LIN {X 0,Y 502.812,Z 410.918,A -85,B 0,C 180,E1 -5734.96,E2 -5734.96} C_VEL
LIN {X 0,Y 504.611,Z 420.54,A -85,B 0,C 180,E1 -5736.546,E2 -5736.546} C_VEL
LIN {X 0,Y 504.361,Z 436.32,A -85,B 0,C 180,E1 -5739.005,E2 -5739.005} C_VEL
LIN {X 0,Y 503.884,Z 455.526,A -85,B 0,C 180,E1 -5741.972,E2 -5741.972} C_VEL
LIN {X 0,Y 503.523,Z 470.549,A -85,B 0,C 180,E1 -5744.274,E2 -5744.274} C_VEL
LIN {X 0,Y 505.329,Z 482.17,A -85,B 0,C 180,E1 -5744.511,E2 -5744.511} C_VEL
LIN {X 0,Y 504.68,Z 580.109,A -85,B 0,C 180,E1 -5745.998,E2 -5745.998} C_VEL
LIN {X 0,Y 504.442,Z 593.546,A -85,B 0,C 180,E1 -5746.376,E2 -5746.376} C_VEL
LIN {X 0,Y 504.146,Z 606.339,A -85,B 0,C 180,E1 -5746.907,E2 -5746.907} C_VEL
LIN {X 0,Y 503.865,Z 618.187,A -85,B 0,C 180,E1 -5747.573,E2 -5747.573} C_VEL
LIN {X 0,Y 503.569,Z 628.743,A -85,B 0,C 180,E1 -5748.324,E2 -5748.324} C_VEL
LIN {X 0,Y 503.221,Z 639.022,A -85,B 0,C 180,E1 -5749.234,E2 -5749.234} C_VEL
LIN {X 0,Y 502.902,Z 649.127,A -85,B 0,C 180,E1 -5750.346,E2 -5750.346} C_VEL
LIN {X 0,Y 502.609,Z 657.945,A -85,B 0,C 180,E1 -5751.557,E2 -5751.557} C_VEL
LIN {X 0,Y 502.408,Z 665.014,A -85,B 0,C 180,E1 -5752.767,E2 -5752.767} C_VEL
LIN {X 0,Y 502.316,Z 670.67,A -85,B 0,C 180,E1 -5753.977,E2 -5753.977} C_VEL
LIN {X 0,Y 502.118,Z 675.083,A -85,B 0,C 180,E1 -5755.183,E2 -5755.183} C_VEL
LIN {X 0,Y 502.218,Z 677.414,A -85,B 0,C 180,E1 -5755.988,E2 -5755.988} C_VEL
LIN {X 0,Y 502.124,Z 679.291,A -85,B 0,C 180,E1 -5756.791,E2 -5756.791} C_VEL
LIN {X 0,Y 502.121,Z 680.748,A -85,B 0,C 180,E1 -5757.593,E2 -5757.593} C_VEL
LIN {X 0,Y 502.036,Z 681.79,A -85,B 0,C 180,E1 -5758.396,E2 -5758.396} C_VEL
LIN {X 0,Y 501.98,Z 682.648,A -85,B 0,C 180,E1 -5760,E2 -5760} C_VEL
LIN {X 0,Y 501.99,Z 682.478,A -85,B 0,C 180,E1 -5760.802,E2 -5760.802} C_VEL
LIN {X 0,Y 502.037,Z 681.897,A -85,B 0,C 180,E1 -5761.604,E2 -5761.604} C_VEL
LIN {X 0,Y 502.121,Z 680.912,A -85,B 0,C 180,E1 -5762.407,E2 -5762.407} C_VEL
LIN {X 0,Y 502.125,Z 679.521,A -85,B 0,C 180,E1 -5763.209,E2 -5763.209} C_VEL
LIN {X 0,Y 502.188,Z 676.607,A -85,B 0,C 180,E1 -5764.414,E2 -5764.414} C_VEL
LIN {X 0,Y 502.289,Z 672.64,A -85,B 0,C 180,E1 -5765.621,E2 -5765.621} C_VEL
LIN {X 0,Y 502.369,Z 666.641,A -85,B 0,C 180,E1 -5767.011,E2 -5767.011} C_VEL
LIN {X 0,Y 502.552,Z 659.852,A -85,B 0,C 180,E1 -5768.241,E2 -5768.241} C_VEL
LIN {X 0,Y 502.792,Z 651.442,A -85,B 0,C 180,E1 -5769.453,E2 -5769.453} C_VEL
LIN {X 0,Y 503.042,Z 642.838,A -85,B 0,C 180,E1 -5770.464,E2 -5770.464} C_VEL
LIN {X 0,Y 503.426,Z 632.166,A -85,B 0,C 180,E1 -5771.475,E2 -5771.475} C_VEL
LIN {X 0,Y 503.752,Z 621.087,A -85,B 0,C 180,E1 -5772.316,E2 -5772.316} C_VEL
LIN {X 0,Y 504.055,Z 609.692,A -85,B 0,C 180,E1 -5772.993,E2 -5772.993} C_VEL
LIN {X 0,Y 504.289,Z 597.377,A -85,B 0,C 180,E1 -5773.551,E2 -5773.551} C_VEL
LIN {X 0,Y 504.521,Z 584.764,A -85,B 0,C 180,E1 -5773.955,E2 -5773.955} C_VEL
LIN {X 0,Y 504.744,Z 570.118,A -85,B 0,C 180,E1 -5774.232,E2 -5774.232} C_VEL
LIN {X 0,Y 505.211,Z 480.854,A -85,B 0,C 180,E1 -5775.591,E2 -5775.591} C_VEL
LIN {X 0,Y 503.576,Z 470.754,A -85,B 0,C 180,E1 -5775.817,E2 -5775.817} C_VEL
LIN {X 0,Y 503.993,Z 450.167,A -85,B 0,C 180,E1 -5778.918,E2 -5778.918} C_VEL
LIN {X 0,Y 504.321,Z 430.326,A -85,B 0,C 180,E1 -5781.887,E2 -5781.887} C_VEL
LIN {X 0,Y 504.447,Z 419.832,A -85,B 0,C 180,E1 -5783.429,E2 -5783.429} C_VEL
LIN {X 0,Y 502.802,Z 410.856,A -85,B 0,C 180,E1 -5784.848,E2 -5784.848} C_VEL
LIN {X 0,Y 502.779,Z 410.86,A -85,B 0,C 180,E1 -5787.47,E2 -5787.47} C_VEL
LIN {X 0,Y 502.805,Z 410.855,A -85,B 0,C 180,E1 -5790.212,E2 -5790.212} C_VEL
LIN {X 0,Y 502.834,Z 410.851,A -85,B 0,C 180,E1 -5793.031,E2 -5793.031} C_VEL
LIN {X 0,Y 502.77,Z 410.856,A -85,B 0,C 180,E1 -5795.952,E2 -5795.952} C_VEL
LIN {X 0,Y 502.803,Z 410.855,A -85,B 0,C 180,E1 -5798.976,E2 -5798.976} C_VEL
LIN {X 0,Y 502.798,Z 410.852,A -85,B 0,C 180,E1 -5802.139,E2 -5802.139} C_VEL
LIN {X 0,Y 502.804,Z 410.854,A -85,B 0,C 180,E1 -5805.468,E2 -5805.468} C_VEL
LIN {X 0,Y 502.822,Z 410.853,A -85,B 0,C 180,E1 -5808.934,E2 -5808.934} C_VEL
LIN {X 0,Y 502.793,Z 410.852,A -85,B 0,C 180,E1 -5812.046,E2 -5812.046} C_VEL
LIN {X 0,Y 502.8,Z 410.854,A -85,B 0,C 180,E1 -5815.034,E2 -5815.034} C_VEL
LIN {X 0,Y 502.785,Z 410.855,A -85,B 0,C 180,E1 -5817.915,E2 -5817.915} C_VEL
LIN {X 0,Y 502.806,Z 410.856,A -85,B 0,C 180,E1 -5820.711,E2 -5820.711} C_VEL
LIN {X 0,Y 502.835,Z 411.023,A -85,B 0,C 180,E1 -5822.336,E2 -5822.336} C_VEL
LIN {X 0,Y 505.373,Z 423.463,A -85,B 0,C 180,E1 -5824.241,E2 -5824.241} C_VEL
LIN {X 0,Y 504.875,Z 441.29,A -85,B 0,C 180,E1 -5826.743,E2 -5826.743} C_VEL
LIN {X 0,Y 504.364,Z 458.409,A -85,B 0,C 180,E1 -5829.112,E2 -5829.112} C_VEL
LIN {X 0,Y 503.788,Z 480.465,A -85,B 0,C 180,E1 -5832.127,E2 -5832.127} C_VEL
LIN {X 0,Y 503.365,Z 495.682,A -85,B 0,C 180,E1 -5834.186,E2 -5834.186} C_VEL
LIN {X 0,Y 505.216,Z 510.923,A -85,B 0,C 180,E1 -5834.498,E2 -5834.498} C_VEL
LIN {X 0,Y 504.735,Z 596.683,A -85,B 0,C 180,E1 -5835.768,E2 -5835.768} C_VEL
LIN {X 0,Y 504.502,Z 611.005,A -85,B 0,C 180,E1 -5836.044,E2 -5836.044} C_VEL
LIN {X 0,Y 504.216,Z 624.892,A -85,B 0,C 180,E1 -5836.499,E2 -5836.499} C_VEL
LIN {X 0,Y 503.892,Z 635.855,A -85,B 0,C 180,E1 -5837.003,E2 -5837.003} C_VEL
LIN {X 0,Y 503.617,Z 646.876,A -85,B 0,C 180,E1 -5837.649,E2 -5837.649} C_VEL
LIN {X 0,Y 503.303,Z 657.249,A -85,B 0,C 180,E1 -5838.42,E2 -5838.42} C_VEL
LIN {X 0,Y 502.974,Z 667.319,A -85,B 0,C 180,E1 -5839.331,E2 -5839.331} C_VEL
LIN {X 0,Y 502.708,Z 676.4,A -85,B 0,C 180,E1 -5840.342,E2 -5840.342} C_VEL
LIN {X 0,Y 502.53,Z 683.874,A -85,B 0,C 180,E1 -5841.353,E2 -5841.353} C_VEL
LIN {X 0,Y 502.351,Z 691.292,A -85,B 0,C 180,E1 -5842.564,E2 -5842.564} C_VEL
LIN {X 0,Y 502.235,Z 696.303,A -85,B 0,C 180,E1 -5843.572,E2 -5843.572} C_VEL
LIN {X 0,Y 502.184,Z 701.137,A -85,B 0,C 180,E1 -5844.781,E2 -5844.781} C_VEL
LIN {X 0,Y 502.231,Z 704.816,A -85,B 0,C 180,E1 -5845.988,E2 -5845.988} C_VEL
LIN {X 0,Y 502.206,Z 706.732,A -85,B 0,C 180,E1 -5846.791,E2 -5846.791} C_VEL
LIN {X 0,Y 502.124,Z 708.179,A -85,B 0,C 180,E1 -5847.593,E2 -5847.593} C_VEL
LIN {X 0,Y 502.041,Z 709.755,A -85,B 0,C 180,E1 -5849.198,E2 -5849.198} C_VEL
LIN {X 0,Y 502.04,Z 709.991,A -85,B 0,C 180,E1 -5850,E2 -5850} C_VEL
LIN {X 0,Y 502.041,Z 709.76,A -85,B 0,C 180,E1 -5850.802,E2 -5850.802} C_VEL
LIN {X 0,Y 502.065,Z 709.113,A -85,B 0,C 180,E1 -5851.604,E2 -5851.604} C_VEL
LIN {X 0,Y 502.206,Z 706.61,A -85,B 0,C 180,E1 -5853.209,E2 -5853.209} C_VEL
LIN {X 0,Y 502.202,Z 703.539,A -85,B 0,C 180,E1 -5854.414,E2 -5854.414} C_VEL
LIN {X 0,Y 502.272,Z 699.389,A -85,B 0,C 180,E1 -5855.621,E2 -5855.621} C_VEL
LIN {X 0,Y 502.316,Z 694.249,A -85,B 0,C 180,E1 -5856.79,E2 -5856.79} C_VEL
LIN {X 0,Y 502.403,Z 688.572,A -85,B 0,C 180,E1 -5857.839,E2 -5857.839} C_VEL
LIN {X 0,Y 502.585,Z 682.001,A -85,B 0,C 180,E1 -5858.848,E2 -5858.848} C_VEL
LIN {X 0,Y 502.79,Z 674.116,A -85,B 0,C 180,E1 -5859.859,E2 -5859.859} C_VEL
LIN {X 0,Y 503.073,Z 664.588,A -85,B 0,C 180,E1 -5860.871,E2 -5860.871} C_VEL
LIN {X 0,Y 503.361,Z 655.159,A -85,B 0,C 180,E1 -5861.68,E2 -5861.68} C_VEL
LIN {X 0,Y 503.524,Z 645.309,A -85,B 0,C 180,E1 -5862.381,E2 -5862.381} C_VEL
LIN {X 0,Y 503.86,Z 633.683,A -85,B 0,C 180,E1 -5863.049,E2 -5863.049} C_VEL
LIN {X 0,Y 504.154,Z 622.054,A -85,B 0,C 180,E1 -5863.555,E2 -5863.555} C_VEL
LIN {X 0,Y 504.488,Z 608.94,A -85,B 0,C 180,E1 -5863.956,E2 -5863.956} C_VEL
LIN {X 0,Y 504.652,Z 593.561,A -85,B 0,C 180,E1 -5864.234,E2 -5864.234} C_VEL
LIN {X 0,Y 505.203,Z 510.39,A -85,B 0,C 180,E1 -5865.485,E2 -5865.485} C_VEL
LIN {X 0,Y 503.281,Z 493.921,A -85,B 0,C 180,E1 -5865.828,E2 -5865.828} C_VEL
LIN {X 0,Y 503.793,Z 470.715,A -85,B 0,C 180,E1 -5868.926,E2 -5868.926} C_VEL
LIN {X 0,Y 504.326,Z 447.248,A -85,B 0,C 180,E1 -5872.102,E2 -5872.102} C_VEL
LIN {X 0,Y 504.989,Z 424.658,A -85,B 0,C 180,E1 -5875.228,E2 -5875.228} C_VEL
LIN {X 0,Y 504.522,Z 419.183,A -85,B 0,C 180,E1 -5876.027,E2 -5876.027} C_VEL
LIN {X 0,Y 502.809,Z 410.856,A -85,B 0,C 180,E1 -5877.311,E2 -5877.311} C_VEL
LIN {X 0,Y 502.805,Z 410.856,A -85,B 0,C 180,E1 -5880.212,E2 -5880.212} C_VEL
LIN {X 0,Y 502.834,Z 410.851,A -85,B 0,C 180,E1 -5883.031,E2 -5883.031} C_VEL
LIN {X 0,Y 502.769,Z 410.858,A -85,B 0,C 180,E1 -5885.952,E2 -5885.952} C_VEL
LIN {X 0,Y 502.803,Z 410.854,A -85,B 0,C 180,E1 -5888.976,E2 -5888.976} C_VEL
LIN {X 0,Y 502.805,Z 410.85,A -85,B 0,C 180,E1 -5892.199,E2 -5892.199} C_VEL
LIN {X 0,Y 502.804,Z 410.856,A -85,B 0,C 180,E1 -5895.468,E2 -5895.468} C_VEL
LIN {X 0,Y 502.822,Z 410.853,A -85,B 0,C 180,E1 -5898.934,E2 -5898.934} C_VEL
LIN {X 0,Y 502.796,Z 410.851,A -85,B 0,C 180,E1 -5902.046,E2 -5902.046} C_VEL
LIN {X 0,Y 502.803,Z 410.857,A -85,B 0,C 180,E1 -5905.034,E2 -5905.034} C_VEL
LIN {X 0,Y 502.786,Z 410.853,A -85,B 0,C 180,E1 -5907.915,E2 -5907.915} C_VEL
LIN {X 0,Y 502.825,Z 410.854,A -85,B 0,C 180,E1 -5910.712,E2 -5910.712} C_VEL
LIN {X 0,Y 502.866,Z 410.845,A -85,B 0,C 180,E1 -5913.439,E2 -5913.439} C_VEL
LIN {X 0,Y 502.779,Z 410.858,A -85,B 0,C 180,E1 -5916.086,E2 -5916.086} C_VEL
LIN {X 0,Y 502.786,Z 410.86,A -85,B 0,C 180,E1 -5918.689,E2 -5918.689} C_VEL
LIN {X 0,Y 502.825,Z 410.851,A -85,B 0,C 180,E1 -5921.248,E2 -5921.248} C_VEL
LIN {X 0,Y 502.835,Z 410.853,A -85,B 0,C 180,E1 -5924.345,E2 -5924.345} C_VEL
LIN {X 0,Y 505.443,Z 418.562,A -85,B 0,C 180,E1 -5924.56,E2 -5924.56} C_VEL
LIN {X 0,Y 504.73,Z 513.794,A -85,B 0,C 180,E1 -5926.051,E2 -5926.051} C_VEL
LIN {X 0,Y 504.537,Z 527.27,A -85,B 0,C 180,E1 -5926.43,E2 -5926.43} C_VEL
LIN {X 0,Y 504.305,Z 539.968,A -85,B 0,C 180,E1 -5926.962,E2 -5926.962} C_VEL
LIN {X 0,Y 504.046,Z 551.757,A -85,B 0,C 180,E1 -5927.631,E2 -5927.631} C_VEL
LIN {X 0,Y 503.743,Z 562.812,A -85,B 0,C 180,E1 -5928.431,E2 -5928.431} C_VEL
LIN {X 0,Y 503.456,Z 572.863,A -85,B 0,C 180,E1 -5929.341,E2 -5929.341} C_VEL
LIN {X 0,Y 503.173,Z 581.893,A -85,B 0,C 180,E1 -5930.351,E2 -5930.351} C_VEL
LIN {X 0,Y 502.846,Z 590.669,A -85,B 0,C 180,E1 -5931.561,E2 -5931.561} C_VEL
LIN {X 0,Y 502.642,Z 597.668,A -85,B 0,C 180,E1 -5932.771,E2 -5932.771} C_VEL
LIN {X 0,Y 502.535,Z 603.214,A -85,B 0,C 180,E1 -5933.979,E2 -5933.979} C_VEL
LIN {X 0,Y 502.328,Z 607.57,A -85,B 0,C 180,E1 -5935.185,E2 -5935.185} C_VEL
LIN {X 0,Y 502.363,Z 609.847,A -85,B 0,C 180,E1 -5935.989,E2 -5935.989} C_VEL
LIN {X 0,Y 502.26,Z 611.712,A -85,B 0,C 180,E1 -5936.791,E2 -5936.791} C_VEL
LIN {X 0,Y 502.166,Z 613.13,A -85,B 0,C 180,E1 -5937.594,E2 -5937.594} C_VEL
LIN {X 0,Y 502.085,Z 614.717,A -85,B 0,C 180,E1 -5939.198,E2 -5939.198} C_VEL
LIN {X 0,Y 502.079,Z 614.934,A -85,B 0,C 180,E1 -5940,E2 -5940} C_VEL
LIN {X 0,Y 502.082,Z 614.729,A -85,B 0,C 180,E1 -5940.802,E2 -5940.802} C_VEL
LIN {X 0,Y 502.152,Z 613.119,A -85,B 0,C 180,E1 -5942.406,E2 -5942.406} C_VEL
LIN {X 0,Y 502.256,Z 611.723,A -85,B 0,C 180,E1 -5943.209,E2 -5943.209} C_VEL
LIN {X 0,Y 502.359,Z 608.801,A -85,B 0,C 180,E1 -5944.413,E2 -5944.413} C_VEL
LIN {X 0,Y 502.343,Z 604.86,A -85,B 0,C 180,E1 -5945.62,E2 -5945.62} C_VEL
LIN {X 0,Y 502.52,Z 598.883,A -85,B 0,C 180,E1 -5947.004,E2 -5947.004} C_VEL
LIN {X 0,Y 502.77,Z 592.082,A -85,B 0,C 180,E1 -5948.238,E2 -5948.238} C_VEL
LIN {X 0,Y 502.992,Z 583.786,A -85,B 0,C 180,E1 -5949.449,E2 -5949.449} C_VEL
LIN {X 0,Y 503.332,Z 575.218,A -85,B 0,C 180,E1 -5950.458,E2 -5950.458} C_VEL
LIN {X 0,Y 503.631,Z 564.636,A -85,B 0,C 180,E1 -5951.47,E2 -5951.47} C_VEL
LIN {X 0,Y 503.938,Z 555.004,A -85,B 0,C 180,E1 -5952.216,E2 -5952.216} C_VEL
LIN {X 0,Y 504.182,Z 544.302,A -85,B 0,C 180,E1 -5952.887,E2 -5952.887} C_VEL
LIN {X 0,Y 504.424,Z 532.882,A -85,B 0,C 180,E1 -5953.445,E2 -5953.445} C_VEL
LIN {X 0,Y 504.654,Z 519.828,A -85,B 0,C 180,E1 -5953.9,E2 -5953.9} C_VEL
LIN {X 0,Y 504.785,Z 507.422,A -85,B 0,C 180,E1 -5954.179,E2 -5954.179} C_VEL
LIN {X 0,Y 505.314,Z 418.371,A -85,B 0,C 180,E1 -5955.527,E2 -5955.527} C_VEL
LIN {X 0,Y 502.826,Z 410.854,A -85,B 0,C 180,E1 -5955.73,E2 -5955.73} C_VEL
LIN {X 0,Y 502.814,Z 410.852,A -85,B 0,C 180,E1 -5958.752,E2 -5958.752} C_VEL
LIN {X 0,Y 502.784,Z 410.861,A -85,B 0,C 180,E1 -5961.311,E2 -5961.311} C_VEL
LIN {X 0,Y 502.772,Z 410.854,A -85,B 0,C 180,E1 -5963.915,E2 -5963.915} C_VEL
LIN {X 0,Y 502.839,Z 410.845,A -85,B 0,C 180,E1 -5966.568,E2 -5966.568} C_VEL
LIN {X 0,Y 502.825,Z 410.855,A -85,B 0,C 180,E1 -5969.288,E2 -5969.288} C_VEL
LIN {X 0,Y 502.786,Z 410.848,A -85,B 0,C 180,E1 -5972.085,E2 -5972.085} C_VEL
LIN {X 0,Y 502.802,Z 410.849,A -85,B 0,C 180,E1 -5974.966,E2 -5974.966} C_VEL
LIN {X 0,Y 502.796,Z 410.851,A -85,B 0,C 180,E1 -5977.954,E2 -5977.954} C_VEL
LIN {X 0,Y 502.823,Z 410.85,A -85,B 0,C 180,E1 -5981.066,E2 -5981.066} C_VEL
LIN {X 0,Y 502.767,Z 410.856,A -85,B 0,C 180,E1 -5983.56,E2 -5983.56} C_VEL
LIN {X 0,Y 502.089,Z 410.943,A -85,B 0,C 180,E1 -5984.229,E2 -5984.229} C_VEL
LIN {X 0,Y 499.217,Z 411.293,A -85,B 0,C 180,E1 -5985.314,E2 -5985.314} C_VEL
LIN {X 0,Y 496.809,Z 411.592,A -85,B 0,C 180,E1 -5986.189,E2 -5986.189} C_VEL
LIN {X 0,Y 495.798,Z 411.727,A -85,B 0,C 180,E1 -5986.865,E2 -5986.865} C_VEL
LIN {X 0,Y 495.728,Z 411.735,A -85,B 0,C 180,E1 -5987.094,E2 -5987.094} C_VEL
LIN {X 0,Y 495.761,Z 411.724,A -85,B 0,C 180,E1 -5989.953,E2 -5989.953} C_VEL
LIN {X 0,Y 495.721,Z 411.738,A -85,B 0,C 180,E1 -5992.555,E2 -5992.555} C_VEL
LIN {X 0,Y 495.78,Z 411.725,A -85,B 0,C 180,E1 -5995.457,E2 -5995.457} C_VEL
LIN {X 0,Y 495.757,Z 411.734,A -85,B 0,C 180,E1 -5998.364,E2 -5998.364} C_VEL
LIN {X 0,Y 495.74,Z 411.734,A -85,B 0,C 180,E1 -6001.518,E2 -6001.518} C_VEL
LIN {X 0,Y 495.756,Z 411.755,A -85,B 0,C 180,E1 -6004.775,E2 -6004.775} C_VEL
LIN {X 0,Y 497.706,Z 422.006,A -85,B 0,C 180,E1 -6006.49,E2 -6006.49} C_VEL
LIN {X 0,Y 497.308,Z 438.63,A -85,B 0,C 180,E1 -6009.143,E2 -6009.143} C_VEL
LIN {X 0,Y 496.828,Z 455.991,A -85,B 0,C 180,E1 -6011.868,E2 -6011.868} C_VEL
LIN {X 0,Y 496.586,Z 470.293,A -85,B 0,C 180,E1 -6014.017,E2 -6014.017} C_VEL
LIN {X 0,Y 498.587,Z 482.825,A -85,B 0,C 180,E1 -6014.271,E2 -6014.271} C_VEL
LIN {X 0,Y 497.993,Z 578.618,A -85,B 0,C 180,E1 -6015.675,E2 -6015.675} C_VEL
LIN {X 0,Y 497.758,Z 592.263,A -85,B 0,C 180,E1 -6016.034,E2 -6016.034} C_VEL
LIN {X 0,Y 497.478,Z 604.399,A -85,B 0,C 180,E1 -6016.52,E2 -6016.52} C_VEL
LIN {X 0,Y 497.123,Z 617.014,A -85,B 0,C 180,E1 -6017.208,E2 -6017.208} C_VEL
LIN {X 0,Y 496.84,Z 627.65,A -85,B 0,C 180,E1 -6017.957,E2 -6017.957} C_VEL
LIN {X 0,Y 496.385,Z 638.11,A -85,B 0,C 180,E1 -6018.877,E2 -6018.877} C_VEL
LIN {X 0,Y 495.982,Z 648.406,A -85,B 0,C 180,E1 -6020.004,E2 -6020.004} C_VEL
LIN {X 0,Y 495.678,Z 657.346,A -85,B 0,C 180,E1 -6021.233,E2 -6021.233} C_VEL
LIN {X 0,Y 495.404,Z 664.523,A -85,B 0,C 180,E1 -6022.46,E2 -6022.46} C_VEL
LIN {X 0,Y 495.253,Z 669.395,A -85,B 0,C 180,E1 -6023.481,E2 -6023.481} C_VEL
LIN {X 0,Y 495.128,Z 674.109,A -85,B 0,C 180,E1 -6024.706,E2 -6024.706} C_VEL
LIN {X 0,Y 495.148,Z 677.717,A -85,B 0,C 180,E1 -6025.93,E2 -6025.93} C_VEL
LIN {X 0,Y 495.05,Z 679.577,A -85,B 0,C 180,E1 -6026.745,E2 -6026.745} C_VEL
LIN {X 0,Y 495.025,Z 681.001,A -85,B 0,C 180,E1 -6027.559,E2 -6027.559} C_VEL
LIN {X 0,Y 494.911,Z 682.615,A -85,B 0,C 180,E1 -6029.186,E2 -6029.186} C_VEL
LIN {X 0,Y 494.898,Z 682.853,A -85,B 0,C 180,E1 -6030,E2 -6030} C_VEL
LIN {X 0,Y 494.911,Z 682.667,A -85,B 0,C 180,E1 -6030.814,E2 -6030.814} C_VEL
LIN {X 0,Y 495.025,Z 681.121,A -85,B 0,C 180,E1 -6032.441,E2 -6032.441} C_VEL
LIN {X 0,Y 495.051,Z 679.763,A -85,B 0,C 180,E1 -6033.255,E2 -6033.255} C_VEL
LIN {X 0,Y 495.102,Z 676.905,A -85,B 0,C 180,E1 -6034.478,E2 -6034.478} C_VEL
LIN {X 0,Y 495.234,Z 673.02,A -85,B 0,C 180,E1 -6035.701,E2 -6035.701} C_VEL
LIN {X 0,Y 495.308,Z 667.992,A -85,B 0,C 180,E1 -6036.927,E2 -6036.927} C_VEL
LIN {X 0,Y 495.52,Z 661.646,A -85,B 0,C 180,E1 -6038.154,E2 -6038.154} C_VEL
LIN {X 0,Y 495.766,Z 653.766,A -85,B 0,C 180,E1 -6039.383,E2 -6039.383} C_VEL
LIN {X 0,Y 496.058,Z 645.718,A -85,B 0,C 180,E1 -6040.407,E2 -6040.407} C_VEL
LIN {X 0,Y 496.495,Z 635.844,A -85,B 0,C 180,E1 -6041.43,E2 -6041.43} C_VEL
LIN {X 0,Y 496.888,Z 624.635,A -85,B 0,C 180,E1 -6042.362,E2 -6042.362} C_VEL
LIN {X 0,Y 497.232,Z 613.919,A -85,B 0,C 180,E1 -6043.07,E2 -6043.07} C_VEL
LIN {X 0,Y 497.547,Z 601.827,A -85,B 0,C 180,E1 -6043.686,E2 -6043.686} C_VEL
LIN {X 0,Y 497.877,Z 588.519,A -85,B 0,C 180,E1 -6044.171,E2 -6044.171} C_VEL
LIN {X 0,Y 498.052,Z 576.639,A -85,B 0,C 180,E1 -6044.453,E2 -6044.453} C_VEL
LIN {X 0,Y 498.539,Z 482.079,A -85,B 0,C 180,E1 -6045.832,E2 -6045.832} C_VEL
LIN {X 0,Y 496.57,Z 470.209,A -85,B 0,C 180,E1 -6046.082,E2 -6046.082} C_VEL
LIN {X 0,Y 496.967,Z 451.125,A -85,B 0,C 180,E1 -6048.981,E2 -6048.981} C_VEL
LIN {X 0,Y 497.506,Z 432.156,A -85,B 0,C 180,E1 -6051.984,E2 -6051.984} C_VEL
LIN {X 0,Y 497.746,Z 422.712,A -85,B 0,C 180,E1 -6053.486,E2 -6053.486} C_VEL
LIN {X 0,Y 495.74,Z 411.737,A -85,B 0,C 180,E1 -6055.338,E2 -6055.338} C_VEL
LIN {X 0,Y 495.74,Z 411.732,A -85,B 0,C 180,E1 -6058.482,E2 -6058.482} C_VEL
LIN {X 0,Y 495.757,Z 411.736,A -85,B 0,C 180,E1 -6061.636,E2 -6061.636} C_VEL
LIN {X 0,Y 495.78,Z 411.727,A -85,B 0,C 180,E1 -6064.543,E2 -6064.543} C_VEL
LIN {X 0,Y 495.724,Z 411.737,A -85,B 0,C 180,E1 -6067.562,E2 -6067.562} C_VEL
LIN {X 0,Y 495.769,Z 411.726,A -85,B 0,C 180,E1 -6070.7,E2 -6070.7} C_VEL
LIN {X 0,Y 495.737,Z 411.728,A -85,B 0,C 180,E1 -6074.001,E2 -6074.001} C_VEL
LIN {X 0,Y 495.73,Z 411.734,A -85,B 0,C 180,E1 -6077.117,E2 -6077.117} C_VEL
LIN {X 0,Y 495.762,Z 411.727,A -85,B 0,C 180,E1 -6079.953,E2 -6079.953} C_VEL
LIN {X 0,Y 495.722,Z 411.736,A -85,B 0,C 180,E1 -6082.554,E2 -6082.554} C_VEL
LIN {X 0,Y 495.78,Z 411.724,A -85,B 0,C 180,E1 -6085.457,E2 -6085.457} C_VEL
LIN {X 0,Y 495.757,Z 411.734,A -85,B 0,C 180,E1 -6088.364,E2 -6088.364} C_VEL
LIN {X 0,Y 495.74,Z 411.731,A -85,B 0,C 180,E1 -6091.518,E2 -6091.518} C_VEL
LIN {X 0,Y 495.778,Z 411.816,A -85,B 0,C 180,E1 -6094.776,E2 -6094.776} C_VEL
LIN {X 0,Y 497.561,Z 420.974,A -85,B 0,C 180,E1 -6096.306,E2 -6096.306} C_VEL
LIN {X 0,Y 497.665,Z 427.684,A -85,B 0,C 180,E1 -6097.367,E2 -6097.367} C_VEL
LIN {X 0,Y 497.204,Z 444.245,A -85,B 0,C 180,E1 -6099.954,E2 -6099.954} C_VEL
LIN {X 0,Y 496.748,Z 461.979,A -85,B 0,C 180,E1 -6102.716,E2 -6102.716} C_VEL
LIN {X 0,Y 496.599,Z 470.761,A -85,B 0,C 180,E1 -6104.053,E2 -6104.053} C_VEL
LIN {X 0,Y 498.5,Z 482.776,A -85,B 0,C 180,E1 -6104.306,E2 -6104.306} C_VEL
LIN {X 0,Y 497.776,Z 580.486,A -85,B 0,C 180,E1 -6105.826,E2 -6105.826} C_VEL
LIN {X 0,Y 497.494,Z 593.83,A -85,B 0,C 180,E1 -6106.208,E2 -6106.208} C_VEL
LIN {X 0,Y 497.222,Z 606.079,A -85,B 0,C 180,E1 -6106.721,E2 -6106.721} C_VEL
LIN {X 0,Y 496.876,Z 618.283,A -85,B 0,C 180,E1 -6107.413,E2 -6107.413} C_VEL
LIN {X 0,Y 496.556,Z 629.927,A -85,B 0,C 180,E1 -6108.261,E2 -6108.261} C_VEL
LIN {X 0,Y 496.142,Z 640.999,A -85,B 0,C 180,E1 -6109.285,E2 -6109.285} C_VEL
LIN {X 0,Y 495.799,Z 650.77,A -85,B 0,C 180,E1 -6110.412,E2 -6110.412} C_VEL
LIN {X 0,Y 495.537,Z 659.295,A -85,B 0,C 180,E1 -6111.641,E2 -6111.641} C_VEL
LIN {X 0,Y 495.326,Z 666.262,A -85,B 0,C 180,E1 -6112.889,E2 -6112.889} C_VEL
LIN {X 0,Y 495.229,Z 672.379,A -85,B 0,C 180,E1 -6114.299,E2 -6114.299} C_VEL
LIN {X 0,Y 495.087,Z 676.45,A -85,B 0,C 180,E1 -6115.522,E2 -6115.522} C_VEL
LIN {X 0,Y 495.05,Z 679.461,A -85,B 0,C 180,E1 -6116.745,E2 -6116.745} C_VEL
LIN {X 0,Y 495.025,Z 680.941,A -85,B 0,C 180,E1 -6117.559,E2 -6117.559} C_VEL
LIN {X 0,Y 494.963,Z 681.969,A -85,B 0,C 180,E1 -6118.373,E2 -6118.373} C_VEL
LIN {X 0,Y 494.898,Z 682.854,A -85,B 0,C 180,E1 -6120,E2 -6120} C_VEL
LIN {X 0,Y 494.911,Z 682.668,A -85,B 0,C 180,E1 -6120.814,E2 -6120.814} C_VEL
LIN {X 0,Y 495.025,Z 681.107,A -85,B 0,C 180,E1 -6122.441,E2 -6122.441} C_VEL
LIN {X 0,Y 495.05,Z 679.699,A -85,B 0,C 180,E1 -6123.255,E2 -6123.255} C_VEL
LIN {X 0,Y 495.083,Z 676.773,A -85,B 0,C 180,E1 -6124.478,E2 -6124.478} C_VEL
LIN {X 0,Y 495.254,Z 671.631,A -85,B 0,C 180,E1 -6126.005,E2 -6126.005} C_VEL
LIN {X 0,Y 495.346,Z 665.632,A -85,B 0,C 180,E1 -6127.336,E2 -6127.336} C_VEL
LIN {X 0,Y 495.562,Z 658.619,A -85,B 0,C 180,E1 -6128.564,E2 -6128.564} C_VEL
LIN {X 0,Y 495.845,Z 649.875,A -85,B 0,C 180,E1 -6129.793,E2 -6129.793} C_VEL
LIN {X 0,Y 496.16,Z 639.805,A -85,B 0,C 180,E1 -6130.921,E2 -6130.921} C_VEL
LIN {X 0,Y 496.572,Z 629.61,A -85,B 0,C 180,E1 -6131.842,E2 -6131.842} C_VEL
LIN {X 0,Y 496.877,Z 618.004,A -85,B 0,C 180,E1 -6132.676,E2 -6132.676} C_VEL
LIN {X 0,Y 497.115,Z 606.327,A -85,B 0,C 180,E1 -6133.334,E2 -6133.334} C_VEL
LIN {X 0,Y 497.48,Z 593.273,A -85,B 0,C 180,E1 -6133.87,E2 -6133.87} C_VEL
LIN {X 0,Y 497.706,Z 580.573,A -85,B 0,C 180,E1 -6134.229,E2 -6134.229} C_VEL
LIN {X 0,Y 498.417,Z 481.876,A -85,B 0,C 180,E1 -6135.788,E2 -6135.788} C_VEL
LIN {X 0,Y 496.646,Z 470.915,A -85,B 0,C 180,E1 -6136.049,E2 -6136.049} C_VEL
LIN {X 0,Y 497.053,Z 450.246,A -85,B 0,C 180,E1 -6139.192,E2 -6139.192} C_VEL
LIN {X 0,Y 497.418,Z 431.593,A -85,B 0,C 180,E1 -6141.988,E2 -6141.988} C_VEL
LIN {X 0,Y 497.562,Z 421.413,A -85,B 0,C 180,E1 -6143.517,E2 -6143.517} C_VEL
LIN {X 0,Y 495.752,Z 411.735,A -85,B 0,C 180,E1 -6145.023,E2 -6145.023} C_VEL
LIN {X 0,Y 495.72,Z 411.74,A -85,B 0,C 180,E1 -6147.895,E2 -6147.895} C_VEL
LIN {X 0,Y 495.75,Z 411.733,A -85,B 0,C 180,E1 -6150.688,E2 -6150.688} C_VEL
LIN {X 0,Y 495.761,Z 411.734,A -85,B 0,C 180,E1 -6153.564,E2 -6153.564} C_VEL
LIN {X 0,Y 495.719,Z 411.733,A -85,B 0,C 180,E1 -6156.545,E2 -6156.545} C_VEL
LIN {X 0,Y 495.759,Z 411.731,A -85,B 0,C 180,E1 -6159.638,E2 -6159.638} C_VEL
LIN {X 0,Y 495.74,Z 411.732,A -85,B 0,C 180,E1 -6162.507,E2 -6162.507} C_VEL
LIN {X 0,Y 495.752,Z 411.733,A -85,B 0,C 180,E1 -6165.139,E2 -6165.139} C_VEL
LIN {X 0,Y 495.759,Z 411.73,A -85,B 0,C 180,E1 -6168.219,E2 -6168.219} C_VEL
LIN {X 0,Y 495.752,Z 411.73,A -85,B 0,C 180,E1 -6171.408,E2 -6171.408} C_VEL
LIN {X 0,Y 495.747,Z 411.733,A -85,B 0,C 180,E1 -6174.462,E2 -6174.462} C_VEL
LIN {X 0,Y 495.77,Z 411.727,A -85,B 0,C 180,E1 -6177.406,E2 -6177.406} C_VEL
LIN {X 0,Y 495.759,Z 411.735,A -85,B 0,C 180,E1 -6180.253,E2 -6180.253} C_VEL
LIN {X 0,Y 495.761,Z 411.815,A -85,B 0,C 180,E1 -6182.107,E2 -6182.107} C_VEL
LIN {X 0,Y 498.395,Z 424.455,A -85,B 0,C 180,E1 -6184.078,E2 -6184.078} C_VEL
LIN {X 0,Y 498.172,Z 438.444,A -85,B 0,C 180,E1 -6186.079,E2 -6186.079} C_VEL
LIN {X 0,Y 497.391,Z 459.747,A -85,B 0,C 180,E1 -6189.069,E2 -6189.069} C_VEL
LIN {X 0,Y 496.71,Z 482.987,A -85,B 0,C 180,E1 -6192.29,E2 -6192.29} C_VEL
LIN {X 0,Y 496.36,Z 495.093,A -85,B 0,C 180,E1 -6193.952,E2 -6193.952} C_VEL
LIN {X 0,Y 498.36,Z 511.974,A -85,B 0,C 180,E1 -6194.306,E2 -6194.306} C_VEL
LIN {X 0,Y 497.789,Z 599.815,A -85,B 0,C 180,E1 -6195.643,E2 -6195.643} C_VEL
LIN {X 0,Y 497.512,Z 613.365,A -85,B 0,C 180,E1 -6195.948,E2 -6195.948} C_VEL
LIN {X 0,Y 497.206,Z 626.32,A -85,B 0,C 180,E1 -6196.409,E2 -6196.409} C_VEL
LIN {X 0,Y 496.85,Z 638.695,A -85,B 0,C 180,E1 -6197.023,E2 -6197.023} C_VEL
LIN {X 0,Y 496.511,Z 649.744,A -85,B 0,C 180,E1 -6197.742,E2 -6197.742} C_VEL
LIN {X 0,Y 496.131,Z 660.034,A -85,B 0,C 180,E1 -6198.561,E2 -6198.561} C_VEL
LIN {X 0,Y 495.828,Z 670.325,A -85,B 0,C 180,E1 -6199.588,E2 -6199.588} C_VEL
LIN {X 0,Y 495.568,Z 678.803,A -85,B 0,C 180,E1 -6200.614,E2 -6200.614} C_VEL
LIN {X 0,Y 495.357,Z 687.067,A -85,B 0,C 180,E1 -6201.843,E2 -6201.843} C_VEL
LIN {X 0,Y 495.248,Z 693.65,A -85,B 0,C 180,E1 -6203.072,E2 -6203.072} C_VEL
LIN {X 0,Y 495.181,Z 698.945,A -85,B 0,C 180,E1 -6204.298,E2 -6204.298} C_VEL
LIN {X 0,Y 495.08,Z 703.065,A -85,B 0,C 180,E1 -6205.522,E2 -6205.522} C_VEL
LIN {X 0,Y 495.138,Z 706.063,A -85,B 0,C 180,E1 -6206.745,E2 -6206.745} C_VEL
LIN {X 0,Y 495.06,Z 707.514,A -85,B 0,C 180,E1 -6207.559,E2 -6207.559} C_VEL
LIN {X 0,Y 494.973,Z 709.077,A -85,B 0,C 180,E1 -6209.186,E2 -6209.186} C_VEL
LIN {X 0,Y 494.971,Z 709.326,A -85,B 0,C 180,E1 -6210,E2 -6210} C_VEL
LIN {X 0,Y 494.972,Z 709.09,A -85,B 0,C 180,E1 -6210.814,E2 -6210.814} C_VEL
LIN {X 0,Y 494.997,Z 708.416,A -85,B 0,C 180,E1 -6211.627,E2 -6211.627} C_VEL
LIN {X 0,Y 495.155,Z 705.927,A -85,B 0,C 180,E1 -6213.255,E2 -6213.255} C_VEL
LIN {X 0,Y 495.095,Z 702.941,A -85,B 0,C 180,E1 -6214.478,E2 -6214.478} C_VEL
LIN {X 0,Y 495.164,Z 697.787,A -85,B 0,C 180,E1 -6215.982,E2 -6215.982} C_VEL
LIN {X 0,Y 495.272,Z 691.624,A -85,B 0,C 180,E1 -6217.337,E2 -6217.337} C_VEL
LIN {X 0,Y 495.45,Z 684.499,A -85,B 0,C 180,E1 -6218.566,E2 -6218.566} C_VEL
LIN {X 0,Y 495.672,Z 675.59,A -85,B 0,C 180,E1 -6219.796,E2 -6219.796} C_VEL
LIN {X 0,Y 495.98,Z 666.424,A -85,B 0,C 180,E1 -6220.822,E2 -6220.822} C_VEL
LIN {X 0,Y 496.314,Z 656.194,A -85,B 0,C 180,E1 -6221.745,E2 -6221.745} C_VEL
LIN {X 0,Y 496.553,Z 645.358,A -85,B 0,C 180,E1 -6222.532,E2 -6222.532} C_VEL
LIN {X 0,Y 496.919,Z 632.877,A -85,B 0,C 180,E1 -6223.235,E2 -6223.235} C_VEL
LIN {X 0,Y 497.31,Z 618.443,A -85,B 0,C 180,E1 -6223.823,E2 -6223.823} C_VEL
LIN {X 0,Y 497.633,Z 604.789,A -85,B 0,C 180,E1 -6224.205,E2 -6224.205} C_VEL
LIN {X 0,Y 498.239,Z 510.06,A -85,B 0,C 180,E1 -6225.696,E2 -6225.696} C_VEL
LIN {X 0,Y 496.229,Z 493.172,A -85,B 0,C 180,E1 -6226.045,E2 -6226.045} C_VEL
LIN {X 0,Y 496.787,Z 469.894,A -85,B 0,C 180,E1 -6229.203,E2 -6229.203} C_VEL
LIN {X 0,Y 497.341,Z 448.094,A -85,B 0,C 180,E1 -6232.21,E2 -6232.21} C_VEL
LIN {X 0,Y 498.061,Z 426.114,A -85,B 0,C 180,E1 -6235.309,E2 -6235.309} C_VEL
LIN {X 0,Y 497.816,Z 421.745,A -85,B 0,C 180,E1 -6235.954,E2 -6235.954} C_VEL
LIN {X 0,Y 495.763,Z 411.735,A -85,B 0,C 180,E1 -6237.548,E2 -6237.548} C_VEL
LIN {X 0,Y 495.749,Z 411.734,A -85,B 0,C 180,E1 -6240.688,E2 -6240.688} C_VEL
LIN {X 0,Y 495.761,Z 411.734,A -85,B 0,C 180,E1 -6243.564,E2 -6243.564} C_VEL
LIN {X 0,Y 495.718,Z 411.734,A -85,B 0,C 180,E1 -6246.545,E2 -6246.545} C_VEL
LIN {X 0,Y 495.758,Z 411.733,A -85,B 0,C 180,E1 -6249.638,E2 -6249.638} C_VEL
LIN {X 0,Y 495.737,Z 411.73,A -85,B 0,C 180,E1 -6252.507,E2 -6252.507} C_VEL
LIN {X 0,Y 495.752,Z 411.734,A -85,B 0,C 180,E1 -6255.139,E2 -6255.139} C_VEL
LIN {X 0,Y 495.758,Z 411.727,A -85,B 0,C 180,E1 -6258.219,E2 -6258.219} C_VEL
LIN {X 0,Y 495.753,Z 411.733,A -85,B 0,C 180,E1 -6261.408,E2 -6261.408} C_VEL
LIN {X 0,Y 495.752,Z 411.73,A -85,B 0,C 180,E1 -6264.462,E2 -6264.462} C_VEL
LIN {X 0,Y 495.77,Z 411.73,A -85,B 0,C 180,E1 -6267.406,E2 -6267.406} C_VEL
LIN {X 0,Y 495.769,Z 411.729,A -85,B 0,C 180,E1 -6270.254,E2 -6270.254} C_VEL
LIN {X 0,Y 495.826,Z 411.724,A -85,B 0,C 180,E1 -6273.251,E2 -6273.251} C_VEL
LIN {X 0,Y 495.746,Z 411.738,A -85,B 0,C 180,E1 -6276.613,E2 -6276.613} C_VEL
LIN {X 0,Y 495.782,Z 411.728,A -85,B 0,C 180,E1 -6279.324,E2 -6279.324} C_VEL
LIN {X 0,Y 495.782,Z 411.729,A -85,B 0,C 180,E1 -6281.828,E2 -6281.828} C_VEL
LIN {X 0,Y 495.796,Z 411.729,A -85,B 0,C 180,E1 -6284.116,E2 -6284.116} C_VEL
LIN {X 0,Y 498.634,Z 420.066,A -85,B 0,C 180,E1 -6284.355,E2 -6284.355} C_VEL
LIN {X 0,Y 497.823,Z 514.767,A -85,B 0,C 180,E1 -6285.879,E2 -6285.879} C_VEL
LIN {X 0,Y 497.641,Z 528.129,A -85,B 0,C 180,E1 -6286.265,E2 -6286.265} C_VEL
LIN {X 0,Y 497.416,Z 540.276,A -85,B 0,C 180,E1 -6286.779,E2 -6286.779} C_VEL
LIN {X 0,Y 497.115,Z 552.524,A -85,B 0,C 180,E1 -6287.481,E2 -6287.481} C_VEL
LIN {X 0,Y 496.811,Z 563.249,A -85,B 0,C 180,E1 -6288.267,E2 -6288.267} C_VEL
LIN {X 0,Y 496.507,Z 573.368,A -85,B 0,C 180,E1 -6289.19,E2 -6289.19} C_VEL
LIN {X 0,Y 496.192,Z 582.443,A -85,B 0,C 180,E1 -6290.214,E2 -6290.214} C_VEL
LIN {X 0,Y 495.849,Z 591.256,A -85,B 0,C 180,E1 -6291.441,E2 -6291.441} C_VEL
LIN {X 0,Y 495.625,Z 598.294,A -85,B 0,C 180,E1 -6292.668,E2 -6292.668} C_VEL
LIN {X 0,Y 495.509,Z 603.861,A -85,B 0,C 180,E1 -6293.894,E2 -6293.894} C_VEL
LIN {X 0,Y 495.293,Z 608.232,A -85,B 0,C 180,E1 -6295.116,E2 -6295.116} C_VEL
LIN {X 0,Y 495.328,Z 610.515,A -85,B 0,C 180,E1 -6295.932,E2 -6295.932} C_VEL
LIN {X 0,Y 495.21,Z 612.385,A -85,B 0,C 180,E1 -6296.746,E2 -6296.746} C_VEL
LIN {X 0,Y 495.105,Z 613.809,A -85,B 0,C 180,E1 -6297.559,E2 -6297.559} C_VEL
LIN {X 0,Y 495.018,Z 615.396,A -85,B 0,C 180,E1 -6299.187,E2 -6299.187} C_VEL
LIN {X 0,Y 495.012,Z 615.608,A -85,B 0,C 180,E1 -6300,E2 -6300} C_VEL
LIN {X 0,Y 495.015,Z 615.396,A -85,B 0,C 180,E1 -6300.814,E2 -6300.814} C_VEL
LIN {X 0,Y 495.088,Z 613.77,A -85,B 0,C 180,E1 -6302.441,E2 -6302.441} C_VEL
LIN {X 0,Y 495.206,Z 612.36,A -85,B 0,C 180,E1 -6303.254,E2 -6303.254} C_VEL
LIN {X 0,Y 495.322,Z 609.416,A -85,B 0,C 180,E1 -6304.476,E2 -6304.476} C_VEL
LIN {X 0,Y 495.301,Z 605.449,A -85,B 0,C 180,E1 -6305.7,E2 -6305.7} C_VEL
LIN {X 0,Y 495.503,Z 599.569,A -85,B 0,C 180,E1 -6307.077,E2 -6307.077} C_VEL
LIN {X 0,Y 495.753,Z 592.599,A -85,B 0,C 180,E1 -6308.355,E2 -6308.355} C_VEL
LIN {X 0,Y 495.998,Z 584.252,A -85,B 0,C 180,E1 -6309.584,E2 -6309.584} C_VEL
LIN {X 0,Y 496.352,Z 575.628,A -85,B 0,C 180,E1 -6310.607,E2 -6310.607} C_VEL
LIN {X 0,Y 496.681,Z 564.988,A -85,B 0,C 180,E1 -6311.633,E2 -6311.633} C_VEL
LIN {X 0,Y 497.052,Z 553.921,A -85,B 0,C 180,E1 -6312.486,E2 -6312.486} C_VEL
LIN {X 0,Y 497.281,Z 542.605,A -85,B 0,C 180,E1 -6313.173,E2 -6313.173} C_VEL
LIN {X 0,Y 497.549,Z 530.345,A -85,B 0,C 180,E1 -6313.738,E2 -6313.738} C_VEL
LIN {X 0,Y 497.827,Z 516.888,A -85,B 0,C 180,E1 -6314.173,E2 -6314.173} C_VEL
LIN {X 0,Y 497.967,Z 503.502,A -85,B 0,C 180,E1 -6314.43,E2 -6314.43} C_VEL
LIN {X 0,Y 498.482,Z 419.764,A -85,B 0,C 180,E1 -6315.724,E2 -6315.724} C_VEL
LIN {X 0,Y 495.764,Z 411.733,A -85,B 0,C 180,E1 -6315.952,E2 -6315.952} C_VEL
LIN {X 0,Y 495.775,Z 411.731,A -85,B 0,C 180,E1 -6319.029,E2 -6319.029} C_VEL
LIN {X 0,Y 495.744,Z 411.734,A -85,B 0,C 180,E1 -6321.629,E2 -6321.629} C_VEL
LIN {X 0,Y 495.718,Z 411.731,A -85,B 0,C 180,E1 -6324.277,E2 -6324.277} C_VEL
LIN {X 0,Y 495.785,Z 411.727,A -85,B 0,C 180,E1 -6326.976,E2 -6326.976} C_VEL
LIN {X 0,Y 495.769,Z 411.728,A -85,B 0,C 180,E1 -6329.746,E2 -6329.746} C_VEL
LIN {X 0,Y 495.771,Z 411.723,A -85,B 0,C 180,E1 -6332.594,E2 -6332.594} C_VEL
LIN {X 0,Y 495.751,Z 411.73,A -85,B 0,C 180,E1 -6335.538,E2 -6335.538} C_VEL
LIN {X 0,Y 495.767,Z 411.733,A -85,B 0,C 180,E1 -6338.768,E2 -6338.768} C_VEL
LIN {X 0,Y 495.759,Z 411.727,A -85,B 0,C 180,E1 -6341.781,E2 -6341.781} C_VEL
LIN {X 0,Y 495.752,Z 411.726,A -85,B 0,C 180,E1 -6345.139,E2 -6345.139} C_VEL
LIN {X 0,Y 495.728,Z 411.735,A -85,B 0,C 180,E1 -6347.094,E2 -6347.094} C_VEL
LIN {X 0,Y 495.088,Z 411.82,A -85,B 0,C 180,E1 -6347.771,E2 -6347.771} C_VEL
LIN {X 0,Y 492.227,Z 412.171,A -85,B 0,C 180,E1 -6348.871,E2 -6348.871} C_VEL
LIN {X 0,Y 489.801,Z 412.468,A -85,B 0,C 180,E1 -6349.758,E2 -6349.758} C_VEL
LIN {X 0,Y 488.774,Z 412.599,A -85,B 0,C 180,E1 -6350.443,E2 -6350.443} C_VEL
LIN {X 0,Y 488.7,Z 412.61,A -85,B 0,C 180,E1 -6350.675,E2 -6350.675} C_VEL
LIN {X 0,Y 488.672,Z 412.61,A -85,B 0,C 180,E1 -6353.867,E2 -6353.867} C_VEL
LIN {X 0,Y 488.741,Z 412.606,A -85,B 0,C 180,E1 -6356.877,E2 -6356.877} C_VEL
LIN {X 0,Y 488.721,Z 412.608,A -85,B 0,C 180,E1 -6359.78,E2 -6359.78} C_VEL
LIN {X 0,Y 488.7,Z 412.613,A -85,B 0,C 180,E1 -6363.078,E2 -6363.078} C_VEL
LIN {X 0,Y 488.722,Z 412.812,A -85,B 0,C 180,E1 -6364.614,E2 -6364.614} C_VEL
LIN {X 0,Y 490.779,Z 423.46,A -85,B 0,C 180,E1 -6366.418,E2 -6366.418} C_VEL
LIN {X 0,Y 490.339,Z 440.88,A -85,B 0,C 180,E1 -6369.222,E2 -6369.222} C_VEL
LIN {X 0,Y 489.815,Z 458.71,A -85,B 0,C 180,E1 -6372.032,E2 -6372.032} C_VEL
LIN {X 0,Y 489.644,Z 470.513,A -85,B 0,C 180,E1 -6373.79,E2 -6373.79} C_VEL
LIN {X 0,Y 491.742,Z 484.324,A -85,B 0,C 180,E1 -6374.068,E2 -6374.068} C_VEL
LIN {X 0,Y 491.131,Z 578.682,A -85,B 0,C 180,E1 -6375.471,E2 -6375.471} C_VEL
LIN {X 0,Y 490.89,Z 592.383,A -85,B 0,C 180,E1 -6375.834,E2 -6375.834} C_VEL
LIN {X 0,Y 490.569,Z 604.547,A -85,B 0,C 180,E1 -6376.327,E2 -6376.327} C_VEL
LIN {X 0,Y 490.198,Z 617.024,A -85,B 0,C 180,E1 -6377.015,E2 -6377.015} C_VEL
LIN {X 0,Y 489.901,Z 627.821,A -85,B 0,C 180,E1 -6377.784,E2 -6377.784} C_VEL
LIN {X 0,Y 489.395,Z 638.287,A -85,B 0,C 180,E1 -6378.716,E2 -6378.716} C_VEL
LIN {X 0,Y 488.987,Z 648.587,A -85,B 0,C 180,E1 -6379.859,E2 -6379.859} C_VEL
LIN {X 0,Y 488.651,Z 657.53,A -85,B 0,C 180,E1 -6381.106,E2 -6381.106} C_VEL
LIN {X 0,Y 488.346,Z 664.709,A -85,B 0,C 180,E1 -6382.35,E2 -6382.35} C_VEL
LIN {X 0,Y 488.201,Z 670.657,A -85,B 0,C 180,E1 -6383.64,E2 -6383.64} C_VEL
LIN {X 0,Y 487.975,Z 675.631,A -85,B 0,C 180,E1 -6385.043,E2 -6385.043} C_VEL
LIN {X 0,Y 488.049,Z 677.906,A -85,B 0,C 180,E1 -6385.871,E2 -6385.871} C_VEL
LIN {X 0,Y 487.979,Z 679.766,A -85,B 0,C 180,E1 -6386.697,E2 -6386.697} C_VEL
LIN {X 0,Y 487.933,Z 681.19,A -85,B 0,C 180,E1 -6387.523,E2 -6387.523} C_VEL
LIN {X 0,Y 487.834,Z 682.804,A -85,B 0,C 180,E1 -6389.175,E2 -6389.175} C_VEL
LIN {X 0,Y 487.819,Z 683.042,A -85,B 0,C 180,E1 -6390,E2 -6390} C_VEL
LIN {X 0,Y 487.834,Z 682.855,A -85,B 0,C 180,E1 -6390.825,E2 -6390.825} C_VEL
LIN {X 0,Y 487.933,Z 681.308,A -85,B 0,C 180,E1 -6392.477,E2 -6392.477} C_VEL
LIN {X 0,Y 487.979,Z 679.95,A -85,B 0,C 180,E1 -6393.303,E2 -6393.303} C_VEL
LIN {X 0,Y 488.002,Z 677.091,A -85,B 0,C 180,E1 -6394.543,E2 -6394.543} C_VEL
LIN {X 0,Y 488.187,Z 672.14,A -85,B 0,C 180,E1 -6396.066,E2 -6396.066} C_VEL
LIN {X 0,Y 488.293,Z 666.209,A -85,B 0,C 180,E1 -6397.443,E2 -6397.443} C_VEL
LIN {X 0,Y 488.579,Z 659.405,A -85,B 0,C 180,E1 -6398.687,E2 -6398.687} C_VEL
LIN {X 0,Y 488.884,Z 650.892,A -85,B 0,C 180,E1 -6399.934,E2 -6399.934} C_VEL
LIN {X 0,Y 489.297,Z 642.176,A -85,B 0,C 180,E1 -6400.971,E2 -6400.971} C_VEL
LIN {X 0,Y 489.692,Z 632.608,A -85,B 0,C 180,E1 -6401.906,E2 -6401.906} C_VEL
LIN {X 0,Y 490.06,Z 621.349,A -85,B 0,C 180,E1 -6402.787,E2 -6402.787} C_VEL
LIN {X 0,Y 490.419,Z 610.36,A -85,B 0,C 180,E1 -6403.466,E2 -6403.466} C_VEL
LIN {X 0,Y 490.759,Z 598.305,A -85,B 0,C 180,E1 -6404.038,E2 -6404.038} C_VEL
LIN {X 0,Y 491.06,Z 585.819,A -85,B 0,C 180,E1 -6404.452,E2 -6404.452} C_VEL
LIN {X 0,Y 491.251,Z 571.647,A -85,B 0,C 180,E1 -6404.737,E2 -6404.737} C_VEL
LIN {X 0,Y 491.646,Z 482.49,A -85,B 0,C 180,E1 -6406.053,E2 -6406.053} C_VEL
LIN {X 0,Y 489.612,Z 470.172,A -85,B 0,C 180,E1 -6406.331,E2 -6406.331} C_VEL
LIN {X 0,Y 490.019,Z 452.034,A -85,B 0,C 180,E1 -6409.103,E2 -6409.103} C_VEL
LIN {X 0,Y 490.565,Z 433.317,A -85,B 0,C 180,E1 -6412.09,E2 -6412.09} C_VEL
LIN {X 0,Y 490.79,Z 423.685,A -85,B 0,C 180,E1 -6413.638,E2 -6413.638} C_VEL
LIN {X 0,Y 488.722,Z 412.612,A -85,B 0,C 180,E1 -6415.524,E2 -6415.524} C_VEL
LIN {X 0,Y 488.687,Z 412.61,A -85,B 0,C 180,E1 -6418.685,E2 -6418.685} C_VEL
LIN {X 0,Y 488.692,Z 412.613,A -85,B 0,C 180,E1 -6421.18,E2 -6421.18} C_VEL
LIN {X 0,Y 488.733,Z 412.606,A -85,B 0,C 180,E1 -6424.113,E2 -6424.113} C_VEL
LIN {X 0,Y 488.673,Z 412.616,A -85,B 0,C 180,E1 -6427.16,E2 -6427.16} C_VEL
LIN {X 0,Y 488.721,Z 412.602,A -85,B 0,C 180,E1 -6430.345,E2 -6430.345} C_VEL
LIN {X 0,Y 488.69,Z 412.607,A -85,B 0,C 180,E1 -6433.654,E2 -6433.654} C_VEL
LIN {X 0,Y 488.691,Z 412.611,A -85,B 0,C 180,E1 -6436.346,E2 -6436.346} C_VEL
LIN {X 0,Y 488.736,Z 412.603,A -85,B 0,C 180,E1 -6439.677,E2 -6439.677} C_VEL
LIN {X 0,Y 488.674,Z 412.609,A -85,B 0,C 180,E1 -6442.84,E2 -6442.84} C_VEL
LIN {X 0,Y 488.733,Z 412.602,A -85,B 0,C 180,E1 -6445.887,E2 -6445.887} C_VEL
LIN {X 0,Y 488.693,Z 412.613,A -85,B 0,C 180,E1 -6448.82,E2 -6448.82} C_VEL
LIN {X 0,Y 488.698,Z 412.609,A -85,B 0,C 180,E1 -6451.668,E2 -6451.668} C_VEL
LIN {X 0,Y 488.703,Z 412.636,A -85,B 0,C 180,E1 -6454.579,E2 -6454.579} C_VEL
LIN {X 0,Y 490.757,Z 423.649,A -85,B 0,C 180,E1 -6456.424,E2 -6456.424} C_VEL
LIN {X 0,Y 490.483,Z 438.505,A -85,B 0,C 180,E1 -6458.773,E2 -6458.773} C_VEL
LIN {X 0,Y 489.973,Z 457.94,A -85,B 0,C 180,E1 -6461.822,E2 -6461.822} C_VEL
LIN {X 0,Y 489.614,Z 470.725,A -85,B 0,C 180,E1 -6463.821,E2 -6463.821} C_VEL
LIN {X 0,Y 491.593,Z 482.658,A -85,B 0,C 180,E1 -6464.082,E2 -6464.082} C_VEL
LIN {X 0,Y 490.889,Z 579.697,A -85,B 0,C 180,E1 -6465.622,E2 -6465.622} C_VEL
LIN {X 0,Y 490.586,Z 592.636,A -85,B 0,C 180,E1 -6465.984,E2 -6465.984} C_VEL
LIN {X 0,Y 490.305,Z 605.784,A -85,B 0,C 180,E1 -6466.53,E2 -6466.53} C_VEL
LIN {X 0,Y 489.918,Z 617.075,A -85,B 0,C 180,E1 -6467.164,E2 -6467.164} C_VEL
LIN {X 0,Y 489.656,Z 628.522,A -85,B 0,C 180,E1 -6467.988,E2 -6467.988} C_VEL
LIN {X 0,Y 489.217,Z 638.952,A -85,B 0,C 180,E1 -6468.922,E2 -6468.922} C_VEL
LIN {X 0,Y 488.887,Z 649.148,A -85,B 0,C 180,E1 -6470.066,E2 -6470.066} C_VEL
LIN {X 0,Y 488.595,Z 656.717,A -85,B 0,C 180,E1 -6471.105,E2 -6471.105} C_VEL
LIN {X 0,Y 488.317,Z 664.112,A -85,B 0,C 180,E1 -6472.35,E2 -6472.35} C_VEL
LIN {X 0,Y 488.158,Z 670.315,A -85,B 0,C 180,E1 -6473.663,E2 -6473.663} C_VEL
LIN {X 0,Y 487.977,Z 675.383,A -85,B 0,C 180,E1 -6475.043,E2 -6475.043} C_VEL
LIN {X 0,Y 488.034,Z 677.721,A -85,B 0,C 180,E1 -6475.871,E2 -6475.871} C_VEL
LIN {X 0,Y 487.977,Z 679.626,A -85,B 0,C 180,E1 -6476.697,E2 -6476.697} C_VEL
LIN {X 0,Y 487.933,Z 681.119,A -85,B 0,C 180,E1 -6477.523,E2 -6477.523} C_VEL
LIN {X 0,Y 487.892,Z 682.15,A -85,B 0,C 180,E1 -6478.349,E2 -6478.349} C_VEL
LIN {X 0,Y 487.819,Z 683.044,A -85,B 0,C 180,E1 -6480,E2 -6480} C_VEL
LIN {X 0,Y 487.834,Z 682.856,A -85,B 0,C 180,E1 -6480.825,E2 -6480.825} C_VEL
LIN {X 0,Y 487.893,Z 682.266,A -85,B 0,C 180,E1 -6481.651,E2 -6481.651} C_VEL
LIN {X 0,Y 487.933,Z 681.289,A -85,B 0,C 180,E1 -6482.477,E2 -6482.477} C_VEL
LIN {X 0,Y 487.978,Z 679.872,A -85,B 0,C 180,E1 -6483.303,E2 -6483.303} C_VEL
LIN {X 0,Y 487.984,Z 676.931,A -85,B 0,C 180,E1 -6484.543,E2 -6484.543} C_VEL
LIN {X 0,Y 488.174,Z 671.924,A -85,B 0,C 180,E1 -6486.049,E2 -6486.049} C_VEL
LIN {X 0,Y 488.28,Z 665.727,A -85,B 0,C 180,E1 -6487.443,E2 -6487.443} C_VEL
LIN {X 0,Y 488.508,Z 658.673,A -85,B 0,C 180,E1 -6488.688,E2 -6488.688} C_VEL
LIN {X 0,Y 488.832,Z 649.87,A -85,B 0,C 180,E1 -6489.935,E2 -6489.935} C_VEL
LIN {X 0,Y 489.191,Z 639.747,A -85,B 0,C 180,E1 -6491.078,E2 -6491.078} C_VEL
LIN {X 0,Y 489.603,Z 629.465,A -85,B 0,C 180,E1 -6492.013,E2 -6492.013} C_VEL
LIN {X 0,Y 489.9,Z 618.382,A -85,B 0,C 180,E1 -6492.82,E2 -6492.82} C_VEL
LIN {X 0,Y 490.196,Z 605.958,A -85,B 0,C 180,E1 -6493.525,E2 -6493.525} C_VEL
LIN {X 0,Y 490.55,Z 592.71,A -85,B 0,C 180,E1 -6494.07,E2 -6494.07} C_VEL
LIN {X 0,Y 490.821,Z 579.51,A -85,B 0,C 180,E1 -6494.432,E2 -6494.432} C_VEL
LIN {X 0,Y 491.609,Z 482.759,A -85,B 0,C 180,E1 -6495.999,E2 -6495.999} C_VEL
LIN {X 0,Y 489.733,Z 471.135,A -85,B 0,C 180,E1 -6496.284,E2 -6496.284} C_VEL
LIN {X 0,Y 490.141,Z 450.307,A -85,B 0,C 180,E1 -6499.474,E2 -6499.474} C_VEL
LIN {X 0,Y 490.601,Z 430.07,A -85,B 0,C 180,E1 -6502.532,E2 -6502.532} C_VEL
LIN {X 0,Y 490.617,Z 422.628,A -85,B 0,C 180,E1 -6503.647,E2 -6503.647} C_VEL
LIN {X 0,Y 488.692,Z 412.616,A -85,B 0,C 180,E1 -6505.259,E2 -6505.259} C_VEL
LIN {X 0,Y 488.697,Z 412.613,A -85,B 0,C 180,E1 -6508.332,E2 -6508.332} C_VEL
LIN {X 0,Y 488.692,Z 412.616,A -85,B 0,C 180,E1 -6511.18,E2 -6511.18} C_VEL
LIN {X 0,Y 488.732,Z 412.606,A -85,B 0,C 180,E1 -6514.113,E2 -6514.113} C_VEL
LIN {X 0,Y 488.673,Z 412.616,A -85,B 0,C 180,E1 -6517.16,E2 -6517.16} C_VEL
LIN {X 0,Y 488.721,Z 412.605,A -85,B 0,C 180,E1 -6520.345,E2 -6520.345} C_VEL
LIN {X 0,Y 488.69,Z 412.611,A -85,B 0,C 180,E1 -6523.654,E2 -6523.654} C_VEL
LIN {X 0,Y 488.69,Z 412.611,A -85,B 0,C 180,E1 -6526.346,E2 -6526.346} C_VEL
LIN {X 0,Y 488.735,Z 412.603,A -85,B 0,C 180,E1 -6529.677,E2 -6529.677} C_VEL
LIN {X 0,Y 488.673,Z 412.614,A -85,B 0,C 180,E1 -6532.84,E2 -6532.84} C_VEL
LIN {X 0,Y 488.732,Z 412.604,A -85,B 0,C 180,E1 -6535.887,E2 -6535.887} C_VEL
LIN {X 0,Y 488.692,Z 412.614,A -85,B 0,C 180,E1 -6538.82,E2 -6538.82} C_VEL
LIN {X 0,Y 488.715,Z 412.771,A -85,B 0,C 180,E1 -6541.903,E2 -6541.903} C_VEL
LIN {X 0,Y 491.354,Z 425.158,A -85,B 0,C 180,E1 -6543.865,E2 -6543.865} C_VEL
LIN {X 0,Y 491.535,Z 430.116,A -85,B 0,C 180,E1 -6544.599,E2 -6544.599} C_VEL
LIN {X 0,Y 490.896,Z 445.53,A -85,B 0,C 180,E1 -6546.814,E2 -6546.814} C_VEL
LIN {X 0,Y 490.409,Z 460.941,A -85,B 0,C 180,E1 -6549.006,E2 -6549.006} C_VEL
LIN {X 0,Y 489.68,Z 483.965,A -85,B 0,C 180,E1 -6552.243,E2 -6552.243} C_VEL
LIN {X 0,Y 489.341,Z 494.66,A -85,B 0,C 180,E1 -6553.734,E2 -6553.734} C_VEL
LIN {X 0,Y 491.52,Z 512.78,A -85,B 0,C 180,E1 -6554.104,E2 -6554.104} C_VEL
LIN {X 0,Y 490.767,Z 602.501,A -85,B 0,C 180,E1 -6555.513,E2 -6555.513} C_VEL
LIN {X 0,Y 490.539,Z 615.533,A -85,B 0,C 180,E1 -6555.85,E2 -6555.85} C_VEL
LIN {X 0,Y 490.15,Z 628.695,A -85,B 0,C 180,E1 -6556.368,E2 -6556.368} C_VEL
LIN {X 0,Y 489.75,Z 643.063,A -85,B 0,C 180,E1 -6557.149,E2 -6557.149} C_VEL
LIN {X 0,Y 489.38,Z 654.744,A -85,B 0,C 180,E1 -6557.981,E2 -6557.981} C_VEL
LIN {X 0,Y 489.062,Z 664.139,A -85,B 0,C 180,E1 -6558.814,E2 -6558.814} C_VEL
LIN {X 0,Y 488.723,Z 673.746,A -85,B 0,C 180,E1 -6559.854,E2 -6559.854} C_VEL
LIN {X 0,Y 488.439,Z 681.586,A -85,B 0,C 180,E1 -6560.893,E2 -6560.893} C_VEL
LIN {X 0,Y 488.233,Z 689.214,A -85,B 0,C 180,E1 -6562.14,E2 -6562.14} C_VEL
LIN {X 0,Y 488.061,Z 695.88,A -85,B 0,C 180,E1 -6563.51,E2 -6563.51} C_VEL
LIN {X 0,Y 488.042,Z 700.164,A -85,B 0,C 180,E1 -6564.629,E2 -6564.629} C_VEL
LIN {X 0,Y 488.047,Z 703.852,A -85,B 0,C 180,E1 -6565.871,E2 -6565.871} C_VEL
LIN {X 0,Y 488.058,Z 705.751,A -85,B 0,C 180,E1 -6566.698,E2 -6566.698} C_VEL
LIN {X 0,Y 487.969,Z 707.183,A -85,B 0,C 180,E1 -6567.524,E2 -6567.524} C_VEL
LIN {X 0,Y 487.892,Z 708.81,A -85,B 0,C 180,E1 -6569.175,E2 -6569.175} C_VEL
LIN {X 0,Y 487.888,Z 709.034,A -85,B 0,C 180,E1 -6570,E2 -6570} C_VEL
LIN {X 0,Y 487.891,Z 708.822,A -85,B 0,C 180,E1 -6570.825,E2 -6570.825} C_VEL
LIN {X 0,Y 487.97,Z 707.185,A -85,B 0,C 180,E1 -6572.476,E2 -6572.476} C_VEL
LIN {X 0,Y 488.073,Z 705.754,A -85,B 0,C 180,E1 -6573.302,E2 -6573.302} C_VEL
LIN {X 0,Y 487.993,Z 702.766,A -85,B 0,C 180,E1 -6574.543,E2 -6574.543} C_VEL
LIN {X 0,Y 488.095,Z 698.711,A -85,B 0,C 180,E1 -6575.785,E2 -6575.785} C_VEL
LIN {X 0,Y 488.181,Z 692.451,A -85,B 0,C 180,E1 -6577.237,E2 -6577.237} C_VEL
LIN {X 0,Y 488.365,Z 685.618,A -85,B 0,C 180,E1 -6578.482,E2 -6578.482} C_VEL
LIN {X 0,Y 488.536,Z 678.619,A -85,B 0,C 180,E1 -6579.523,E2 -6579.523} C_VEL
LIN {X 0,Y 488.825,Z 670.155,A -85,B 0,C 180,E1 -6580.563,E2 -6580.563} C_VEL
LIN {X 0,Y 489.156,Z 659.664,A -85,B 0,C 180,E1 -6581.604,E2 -6581.604} C_VEL
LIN {X 0,Y 489.481,Z 649.251,A -85,B 0,C 180,E1 -6582.437,E2 -6582.437} C_VEL
LIN {X 0,Y 489.881,Z 637.734,A -85,B 0,C 180,E1 -6583.164,E2 -6583.164} C_VEL
LIN {X 0,Y 490.181,Z 625.714,A -85,B 0,C 180,E1 -6583.737,E2 -6583.737} C_VEL
LIN {X 0,Y 490.496,Z 612.628,A -85,B 0,C 180,E1 -6584.177,E2 -6584.177} C_VEL
LIN {X 0,Y 490.777,Z 597.341,A -85,B 0,C 180,E1 -6584.513,E2 -6584.513} C_VEL
LIN {X 0,Y 491.467,Z 512.079,A -85,B 0,C 180,E1 -6585.868,E2 -6585.868} C_VEL
LIN {X 0,Y 489.196,Z 492.245,A -85,B 0,C 180,E1 -6586.296,E2 -6586.296} C_VEL
LIN {X 0,Y 489.801,Z 469.168,A -85,B 0,C 180,E1 -6589.488,E2 -6589.488} C_VEL
LIN {X 0,Y 490.429,Z 447.451,A -85,B 0,C 180,E1 -6592.541,E2 -6592.541} C_VEL
LIN {X 0,Y 491.179,Z 425.869,A -85,B 0,C 180,E1 -6595.653,E2 -6595.653} C_VEL
LIN {X 0,Y 490.266,Z 419.968,A -85,B 0,C 180,E1 -6596.575,E2 -6596.575} C_VEL
LIN {X 0,Y 488.721,Z 412.611,A -85,B 0,C 180,E1 -6597.805,E2 -6597.805} C_VEL
LIN {X 0,Y 488.706,Z 412.612,A -85,B 0,C 180,E1 -6600.362,E2 -6600.362} C_VEL
LIN {X 0,Y 488.737,Z 412.609,A -85,B 0,C 180,E1 -6603.484,E2 -6603.484} C_VEL
LIN {X 0,Y 488.675,Z 412.612,A -85,B 0,C 180,E1 -6606.353,E2 -6606.353} C_VEL
LIN {X 0,Y 488.703,Z 412.613,A -85,B 0,C 180,E1 -6609.254,E2 -6609.254} C_VEL
LIN {X 0,Y 488.69,Z 412.608,A -85,B 0,C 180,E1 -6612.526,E2 -6612.526} C_VEL
LIN {X 0,Y 488.715,Z 412.611,A -85,B 0,C 180,E1 -6615.199,E2 -6615.199} C_VEL
LIN {X 0,Y 488.709,Z 412.606,A -85,B 0,C 180,E1 -6618.4,E2 -6618.4} C_VEL
LIN {X 0,Y 488.707,Z 412.613,A -85,B 0,C 180,E1 -6620.947,E2 -6620.947} C_VEL
LIN {X 0,Y 488.68,Z 412.61,A -85,B 0,C 180,E1 -6623.868,E2 -6623.868} C_VEL
LIN {X 0,Y 488.742,Z 412.608,A -85,B 0,C 180,E1 -6626.877,E2 -6626.877} C_VEL
LIN {X 0,Y 488.727,Z 412.605,A -85,B 0,C 180,E1 -6629.781,E2 -6629.781} C_VEL
LIN {X 0,Y 488.794,Z 412.602,A -85,B 0,C 180,E1 -6633.057,E2 -6633.057} C_VEL
LIN {X 0,Y 488.683,Z 412.615,A -85,B 0,C 180,E1 -6636.254,E2 -6636.254} C_VEL
LIN {X 0,Y 488.75,Z 412.605,A -85,B 0,C 180,E1 -6639.176,E2 -6639.176} C_VEL
LIN {X 0,Y 488.75,Z 412.604,A -85,B 0,C 180,E1 -6641.632,E2 -6641.632} C_VEL
LIN {X 0,Y 488.734,Z 412.608,A -85,B 0,C 180,E1 -6643.863,E2 -6643.863} C_VEL
LIN {X 0,Y 491.865,Z 421.959,A -85,B 0,C 180,E1 -6644.15,E2 -6644.15} C_VEL
LIN {X 0,Y 490.928,Z 515.776,A -85,B 0,C 180,E1 -6645.703,E2 -6645.703} C_VEL
LIN {X 0,Y 490.742,Z 529.029,A -85,B 0,C 180,E1 -6646.094,E2 -6646.094} C_VEL
LIN {X 0,Y 490.498,Z 541.62,A -85,B 0,C 180,E1 -6646.641,E2 -6646.641} C_VEL
LIN {X 0,Y 490.195,Z 553.459,A -85,B 0,C 180,E1 -6647.335,E2 -6647.335} C_VEL
LIN {X 0,Y 489.847,Z 565.026,A -85,B 0,C 180,E1 -6648.203,E2 -6648.203} C_VEL
LIN {X 0,Y 489.566,Z 573.93,A -85,B 0,C 180,E1 -6649.035,E2 -6649.035} C_VEL
LIN {X 0,Y 489.229,Z 583.037,A -85,B 0,C 180,E1 -6650.073,E2 -6650.073} C_VEL
LIN {X 0,Y 488.866,Z 591.869,A -85,B 0,C 180,E1 -6651.318,E2 -6651.318} C_VEL
LIN {X 0,Y 488.628,Z 598.931,A -85,B 0,C 180,E1 -6652.562,E2 -6652.562} C_VEL
LIN {X 0,Y 488.486,Z 604.514,A -85,B 0,C 180,E1 -6653.805,E2 -6653.805} C_VEL
LIN {X 0,Y 488.26,Z 608.895,A -85,B 0,C 180,E1 -6655.046,E2 -6655.046} C_VEL
LIN {X 0,Y 488.294,Z 611.184,A -85,B 0,C 180,E1 -6655.873,E2 -6655.873} C_VEL
LIN {X 0,Y 488.162,Z 613.059,A -85,B 0,C 180,E1 -6656.699,E2 -6656.699} C_VEL
LIN {X 0,Y 488.044,Z 614.489,A -85,B 0,C 180,E1 -6657.524,E2 -6657.524} C_VEL
LIN {X 0,Y 487.952,Z 616.073,A -85,B 0,C 180,E1 -6659.175,E2 -6659.175} C_VEL
LIN {X 0,Y 487.944,Z 616.281,A -85,B 0,C 180,E1 -6660,E2 -6660} C_VEL
LIN {X 0,Y 487.948,Z 616.064,A -85,B 0,C 180,E1 -6660.825,E2 -6660.825} C_VEL
LIN {X 0,Y 488.026,Z 614.417,A -85,B 0,C 180,E1 -6662.476,E2 -6662.476} C_VEL
LIN {X 0,Y 488.159,Z 612.995,A -85,B 0,C 180,E1 -6663.301,E2 -6663.301} C_VEL
LIN {X 0,Y 488.269,Z 610.031,A -85,B 0,C 180,E1 -6664.541,E2 -6664.541} C_VEL
LIN {X 0,Y 488.26,Z 606.037,A -85,B 0,C 180,E1 -6665.783,E2 -6665.783} C_VEL
LIN {X 0,Y 488.48,Z 600.212,A -85,B 0,C 180,E1 -6667.16,E2 -6667.16} C_VEL
LIN {X 0,Y 488.758,Z 593.106,A -85,B 0,C 180,E1 -6668.476,E2 -6668.476} C_VEL
LIN {X 0,Y 489.012,Z 584.714,A -85,B 0,C 180,E1 -6669.722,E2 -6669.722} C_VEL
LIN {X 0,Y 489.394,Z 576.036,A -85,B 0,C 180,E1 -6670.76,E2 -6670.76} C_VEL
LIN {X 0,Y 489.731,Z 565.338,A -85,B 0,C 180,E1 -6671.8,E2 -6671.8} C_VEL
LIN {X 0,Y 490.105,Z 554.706,A -85,B 0,C 180,E1 -6672.63,E2 -6672.63} C_VEL
LIN {X 0,Y 490.391,Z 542.765,A -85,B 0,C 180,E1 -6673.362,E2 -6673.362} C_VEL
LIN {X 0,Y 490.668,Z 530.381,A -85,B 0,C 180,E1 -6673.935,E2 -6673.935} C_VEL
LIN {X 0,Y 490.93,Z 517.646,A -85,B 0,C 180,E1 -6674.35,E2 -6674.35} C_VEL
LIN {X 0,Y 491.064,Z 504.446,A -85,B 0,C 180,E1 -6674.61,E2 -6674.61} C_VEL
LIN {X 0,Y 491.598,Z 421.206,A -85,B 0,C 180,E1 -6675.928,E2 -6675.928} C_VEL
LIN {X 0,Y 488.708,Z 412.61,A -85,B 0,C 180,E1 -6676.18,E2 -6676.18} C_VEL
LIN {X 0,Y 488.738,Z 412.611,A -85,B 0,C 180,E1 -6679.314,E2 -6679.314} C_VEL
LIN {X 0,Y 488.7,Z 412.607,A -85,B 0,C 180,E1 -6681.957,E2 -6681.957} C_VEL
LIN {X 0,Y 488.704,Z 412.609,A -85,B 0,C 180,E1 -6685.042,E2 -6685.042} C_VEL
LIN {X 0,Y 488.733,Z 412.606,A -85,B 0,C 180,E1 -6687.398,E2 -6687.398} C_VEL
LIN {X 0,Y 488.713,Z 412.605,A -85,B 0,C 180,E1 -6690.363,E2 -6690.363} C_VEL
LIN {X 0,Y 488.737,Z 412.595,A -85,B 0,C 180,E1 -6693.484,E2 -6693.484} C_VEL
LIN {X 0,Y 488.685,Z 412.609,A -85,B 0,C 180,E1 -6696.355,E2 -6696.355} C_VEL
LIN {X 0,Y 488.704,Z 412.605,A -85,B 0,C 180,E1 -6699.254,E2 -6699.254} C_VEL
LIN {X 0,Y 488.71,Z 412.605,A -85,B 0,C 180,E1 -6701.6,E2 -6701.6} C_VEL
LIN {X 0,Y 488.715,Z 412.608,A -85,B 0,C 180,E1 -6704.801,E2 -6704.801} C_VEL
LIN {X 0,Y 488.695,Z 412.608,A -85,B 0,C 180,E1 -6707.475,E2 -6707.475} C_VEL
LIN {X 0,Y 488.736,Z 412.599,A -85,B 0,C 180,E1 -6709.677,E2 -6709.677} C_VEL
LIN {X 0,Y 488.7,Z 412.61,A -85,B 0,C 180,E1 -6710.675,E2 -6710.675} C_VEL
LIN {X 0,Y 488.052,Z 412.699,A -85,B 0,C 180,E1 -6711.362,E2 -6711.362} C_VEL
LIN {X 0,Y 485.182,Z 413.058,A -85,B 0,C 180,E1 -6712.478,E2 -6712.478} C_VEL
LIN {X 0,Y 482.748,Z 413.356,A -85,B 0,C 180,E1 -6713.377,E2 -6713.377} C_VEL
LIN {X 0,Y 481.713,Z 413.481,A -85,B 0,C 180,E1 -6714.072,E2 -6714.072} C_VEL
LIN {X 0,Y 481.635,Z 413.49,A -85,B 0,C 180,E1 -6714.307,E2 -6714.307} C_VEL
LIN {X 0,Y 481.675,Z 413.483,A -85,B 0,C 180,E1 -6717.326,E2 -6717.326} C_VEL
LIN {X 0,Y 481.669,Z 413.491,A -85,B 0,C 180,E1 -6720.258,E2 -6720.258} C_VEL
LIN {X 0,Y 481.662,Z 413.49,A -85,B 0,C 180,E1 -6723.107,E2 -6723.107} C_VEL
LIN {X 0,Y 481.706,Z 413.597,A -85,B 0,C 180,E1 -6724.404,E2 -6724.404} C_VEL
LIN {X 0,Y 483.786,Z 424.27,A -85,B 0,C 180,E1 -6726.236,E2 -6726.236} C_VEL
LIN {X 0,Y 483.572,Z 436.379,A -85,B 0,C 180,E1 -6728.206,E2 -6728.206} C_VEL
LIN {X 0,Y 482.966,Z 455.882,A -85,B 0,C 180,E1 -6731.329,E2 -6731.329} C_VEL
LIN {X 0,Y 482.681,Z 470.434,A -85,B 0,C 180,E1 -6733.542,E2 -6733.542} C_VEL
LIN {X 0,Y 484.925,Z 484.42,A -85,B 0,C 180,E1 -6733.838,E2 -6733.838} C_VEL
LIN {X 0,Y 484.279,Z 578.768,A -85,B 0,C 180,E1 -6735.261,E2 -6735.261} C_VEL
LIN {X 0,Y 484.028,Z 592.514,A -85,B 0,C 180,E1 -6735.629,E2 -6735.629} C_VEL
LIN {X 0,Y 483.683,Z 604.701,A -85,B 0,C 180,E1 -6736.128,E2 -6736.128} C_VEL
LIN {X 0,Y 483.277,Z 617.52,A -85,B 0,C 180,E1 -6736.847,E2 -6736.847} C_VEL
LIN {X 0,Y 482.965,Z 627.992,A -85,B 0,C 180,E1 -6737.606,E2 -6737.606} C_VEL
LIN {X 0,Y 482.449,Z 638.463,A -85,B 0,C 180,E1 -6738.552,E2 -6738.552} C_VEL
LIN {X 0,Y 481.99,Z 648.768,A -85,B 0,C 180,E1 -6739.711,E2 -6739.711} C_VEL
LIN {X 0,Y 481.638,Z 657.714,A -85,B 0,C 180,E1 -6740.975,E2 -6740.975} C_VEL
LIN {X 0,Y 481.313,Z 664.895,A -85,B 0,C 180,E1 -6742.238,E2 -6742.238} C_VEL
LIN {X 0,Y 481.136,Z 671.197,A -85,B 0,C 180,E1 -6743.634,E2 -6743.634} C_VEL
LIN {X 0,Y 480.912,Z 675.819,A -85,B 0,C 180,E1 -6744.97,E2 -6744.97} C_VEL
LIN {X 0,Y 480.95,Z 678.095,A -85,B 0,C 180,E1 -6745.81,E2 -6745.81} C_VEL
LIN {X 0,Y 480.909,Z 679.955,A -85,B 0,C 180,E1 -6746.649,E2 -6746.649} C_VEL
LIN {X 0,Y 480.846,Z 681.379,A -85,B 0,C 180,E1 -6747.487,E2 -6747.487} C_VEL
LIN {X 0,Y 480.823,Z 682.376,A -85,B 0,C 180,E1 -6748.325,E2 -6748.325} C_VEL
LIN {X 0,Y 480.743,Z 683.231,A -85,B 0,C 180,E1 -6750,E2 -6750} C_VEL
LIN {X 0,Y 480.824,Z 682.459,A -85,B 0,C 180,E1 -6751.675,E2 -6751.675} C_VEL
LIN {X 0,Y 480.909,Z 680.136,A -85,B 0,C 180,E1 -6753.351,E2 -6753.351} C_VEL
LIN {X 0,Y 480.906,Z 677.277,A -85,B 0,C 180,E1 -6754.61,E2 -6754.61} C_VEL
LIN {X 0,Y 481.122,Z 673.386,A -85,B 0,C 180,E1 -6755.869,E2 -6755.869} C_VEL
LIN {X 0,Y 481.196,Z 668.352,A -85,B 0,C 180,E1 -6757.131,E2 -6757.131} C_VEL
LIN {X 0,Y 481.449,Z 662.001,A -85,B 0,C 180,E1 -6758.394,E2 -6758.394} C_VEL
LIN {X 0,Y 481.762,Z 654.112,A -85,B 0,C 180,E1 -6759.658,E2 -6759.658} C_VEL
LIN {X 0,Y 482.094,Z 646.056,A -85,B 0,C 180,E1 -6760.712,E2 -6760.712} C_VEL
LIN {X 0,Y 482.591,Z 636.167,A -85,B 0,C 180,E1 -6761.764,E2 -6761.764} C_VEL
LIN {X 0,Y 483.026,Z 624.76,A -85,B 0,C 180,E1 -6762.736,E2 -6762.736} C_VEL
LIN {X 0,Y 483.397,Z 614.203,A -85,B 0,C 180,E1 -6763.451,E2 -6763.451} C_VEL
LIN {X 0,Y 483.78,Z 602.063,A -85,B 0,C 180,E1 -6764.083,E2 -6764.083} C_VEL
LIN {X 0,Y 484.143,Z 588.683,A -85,B 0,C 180,E1 -6764.582,E2 -6764.582} C_VEL
LIN {X 0,Y 484.355,Z 576.62,A -85,B 0,C 180,E1 -6764.871,E2 -6764.871} C_VEL
LIN {X 0,Y 484.931,Z 483.927,A -85,B 0,C 180,E1 -6766.26,E2 -6766.26} C_VEL
LIN {X 0,Y 482.67,Z 470.448,A -85,B 0,C 180,E1 -6766.545,E2 -6766.545} C_VEL
LIN {X 0,Y 483.06,Z 453.332,A -85,B 0,C 180,E1 -6769.172,E2 -6769.172} C_VEL
LIN {X 0,Y 483.628,Z 434.497,A -85,B 0,C 180,E1 -6772.199,E2 -6772.199} C_VEL
LIN {X 0,Y 483.841,Z 424.764,A -85,B 0,C 180,E1 -6773.779,E2 -6773.779} C_VEL
LIN {X 0,Y 481.669,Z 413.491,A -85,B 0,C 180,E1 -6775.727,E2 -6775.727} C_VEL
LIN {X 0,Y 481.642,Z 413.488,A -85,B 0,C 180,E1 -6778.895,E2 -6778.895} C_VEL
LIN {X 0,Y 481.659,Z 413.487,A -85,B 0,C 180,E1 -6782.189,E2 -6782.189} C_VEL
LIN {X 0,Y 481.69,Z 413.483,A -85,B 0,C 180,E1 -6784.682,E2 -6784.682} C_VEL
LIN {X 0,Y 481.653,Z 413.486,A -85,B 0,C 180,E1 -6788.007,E2 -6788.007} C_VEL
LIN {X 0,Y 481.659,Z 413.487,A -85,B 0,C 180,E1 -6791.042,E2 -6791.042} C_VEL
LIN {X 0,Y 481.663,Z 413.482,A -85,B 0,C 180,E1 -6794.457,E2 -6794.457} C_VEL
LIN {X 0,Y 481.651,Z 413.481,A -85,B 0,C 180,E1 -6797.839,E2 -6797.839} C_VEL
LIN {X 0,Y 481.684,Z 413.487,A -85,B 0,C 180,E1 -6800.651,E2 -6800.651} C_VEL
LIN {X 0,Y 481.625,Z 413.482,A -85,B 0,C 180,E1 -6803.377,E2 -6803.377} C_VEL
LIN {X 0,Y 481.713,Z 413.481,A -85,B 0,C 180,E1 -6806.33,E2 -6806.33} C_VEL
LIN {X 0,Y 481.648,Z 413.486,A -85,B 0,C 180,E1 -6809.418,E2 -6809.418} C_VEL
LIN {X 0,Y 481.654,Z 413.49,A -85,B 0,C 180,E1 -6812.165,E2 -6812.165} C_VEL
LIN {X 0,Y 481.708,Z 413.613,A -85,B 0,C 180,E1 -6814.402,E2 -6814.402} C_VEL
LIN {X 0,Y 483.78,Z 424.437,A -85,B 0,C 180,E1 -6816.237,E2 -6816.237} C_VEL
LIN {X 0,Y 483.693,Z 435.503,A -85,B 0,C 180,E1 -6818.001,E2 -6818.001} C_VEL
LIN {X 0,Y 483.112,Z 455.391,A -85,B 0,C 180,E1 -6821.151,E2 -6821.151} C_VEL
LIN {X 0,Y 482.669,Z 470.811,A -85,B 0,C 180,E1 -6823.587,E2 -6823.587} C_VEL
LIN {X 0,Y 484.789,Z 484.727,A -85,B 0,C 180,E1 -6823.892,E2 -6823.892} C_VEL
LIN {X 0,Y 483.982,Z 580.082,A -85,B 0,C 180,E1 -6825.44,E2 -6825.44} C_VEL
LIN {X 0,Y 483.634,Z 593.634,A -85,B 0,C 180,E1 -6825.832,E2 -6825.832} C_VEL
LIN {X 0,Y 483.37,Z 606.547,A -85,B 0,C 180,E1 -6826.387,E2 -6826.387} C_VEL
LIN {X 0,Y 482.958,Z 618.708,A -85,B 0,C 180,E1 -6827.097,E2 -6827.097} C_VEL
LIN {X 0,Y 482.649,Z 629.722,A -85,B 0,C 180,E1 -6827.917,E2 -6827.917} C_VEL
LIN {X 0,Y 482.183,Z 639.917,A -85,B 0,C 180,E1 -6828.865,E2 -6828.865} C_VEL
LIN {X 0,Y 481.884,Z 649.154,A -85,B 0,C 180,E1 -6829.921,E2 -6829.921} C_VEL
LIN {X 0,Y 481.566,Z 656.76,A -85,B 0,C 180,E1 -6830.974,E2 -6830.974} C_VEL
LIN {X 0,Y 481.257,Z 664.197,A -85,B 0,C 180,E1 -6832.237,E2 -6832.237} C_VEL
LIN {X 0,Y 481.094,Z 670.888,A -85,B 0,C 180,E1 -6833.679,E2 -6833.679} C_VEL
LIN {X 0,Y 480.913,Z 675.523,A -85,B 0,C 180,E1 -6834.97,E2 -6834.97} C_VEL
LIN {X 0,Y 480.934,Z 677.876,A -85,B 0,C 180,E1 -6835.81,E2 -6835.81} C_VEL
LIN {X 0,Y 480.907,Z 679.792,A -85,B 0,C 180,E1 -6836.649,E2 -6836.649} C_VEL
LIN {X 0,Y 480.846,Z 681.294,A -85,B 0,C 180,E1 -6837.487,E2 -6837.487} C_VEL
LIN {X 0,Y 480.823,Z 682.331,A -85,B 0,C 180,E1 -6838.325,E2 -6838.325} C_VEL
LIN {X 0,Y 480.743,Z 683.233,A -85,B 0,C 180,E1 -6840,E2 -6840} C_VEL
LIN {X 0,Y 480.76,Z 683.045,A -85,B 0,C 180,E1 -6840.838,E2 -6840.838} C_VEL
LIN {X 0,Y 480.824,Z 682.452,A -85,B 0,C 180,E1 -6841.675,E2 -6841.675} C_VEL
LIN {X 0,Y 480.846,Z 681.472,A -85,B 0,C 180,E1 -6842.513,E2 -6842.513} C_VEL
LIN {X 0,Y 480.907,Z 680.045,A -85,B 0,C 180,E1 -6843.351,E2 -6843.351} C_VEL
LIN {X 0,Y 480.891,Z 677.088,A -85,B 0,C 180,E1 -6844.61,E2 -6844.61} C_VEL
LIN {X 0,Y 481.094,Z 673.057,A -85,B 0,C 180,E1 -6845.869,E2 -6845.869} C_VEL
LIN {X 0,Y 481.196,Z 666.875,A -85,B 0,C 180,E1 -6847.342,E2 -6847.342} C_VEL
LIN {X 0,Y 481.433,Z 660.042,A -85,B 0,C 180,E1 -6848.605,E2 -6848.605} C_VEL
LIN {X 0,Y 481.742,Z 651.504,A -85,B 0,C 180,E1 -6849.87,E2 -6849.87} C_VEL
LIN {X 0,Y 482.058,Z 642.735,A -85,B 0,C 180,E1 -6850.925,E2 -6850.925} C_VEL
LIN {X 0,Y 482.536,Z 631.84,A -85,B 0,C 180,E1 -6851.979,E2 -6851.979} C_VEL
LIN {X 0,Y 482.843,Z 621.594,A -85,B 0,C 180,E1 -6852.782,E2 -6852.782} C_VEL
LIN {X 0,Y 483.19,Z 610.736,A -85,B 0,C 180,E1 -6853.457,E2 -6853.457} C_VEL
LIN {X 0,Y 483.479,Z 598.589,A -85,B 0,C 180,E1 -6854.039,E2 -6854.039} C_VEL
LIN {X 0,Y 483.795,Z 585.423,A -85,B 0,C 180,E1 -6854.485,E2 -6854.485} C_VEL
LIN {X 0,Y 484.042,Z 571.15,A -85,B 0,C 180,E1 -6854.773,E2 -6854.773} C_VEL
LIN {X 0,Y 484.888,Z 484.066,A -85,B 0,C 180,E1 -6856.216,E2 -6856.216} C_VEL
LIN {X 0,Y 482.791,Z 471.381,A -85,B 0,C 180,E1 -6856.534,E2 -6856.534} C_VEL
LIN {X 0,Y 483.239,Z 451.851,A -85,B 0,C 180,E1 -6859.542,E2 -6859.542} C_VEL
LIN {X 0,Y 483.71,Z 431.442,A -85,B 0,C 180,E1 -6862.646,E2 -6862.646} C_VEL
LIN {X 0,Y 483.768,Z 424.205,A -85,B 0,C 180,E1 -6863.76,E2 -6863.76} C_VEL
LIN {X 0,Y 481.669,Z 413.491,A -85,B 0,C 180,E1 -6865.499,E2 -6865.499} C_VEL
LIN {X 0,Y 481.662,Z 413.489,A -85,B 0,C 180,E1 -6868.784,E2 -6868.784} C_VEL
LIN {X 0,Y 481.659,Z 413.487,A -85,B 0,C 180,E1 -6872.189,E2 -6872.189} C_VEL
LIN {X 0,Y 481.69,Z 413.483,A -85,B 0,C 180,E1 -6874.682,E2 -6874.682} C_VEL
LIN {X 0,Y 481.653,Z 413.486,A -85,B 0,C 180,E1 -6878.007,E2 -6878.007} C_VEL
LIN {X 0,Y 481.659,Z 413.489,A -85,B 0,C 180,E1 -6881.042,E2 -6881.042} C_VEL
LIN {X 0,Y 481.662,Z 413.487,A -85,B 0,C 180,E1 -6884.457,E2 -6884.457} C_VEL
LIN {X 0,Y 481.65,Z 413.487,A -85,B 0,C 180,E1 -6887.839,E2 -6887.839} C_VEL
LIN {X 0,Y 481.682,Z 413.485,A -85,B 0,C 180,E1 -6890.651,E2 -6890.651} C_VEL
LIN {X 0,Y 481.624,Z 413.49,A -85,B 0,C 180,E1 -6893.377,E2 -6893.377} C_VEL
LIN {X 0,Y 481.712,Z 413.481,A -85,B 0,C 180,E1 -6896.33,E2 -6896.33} C_VEL
LIN {X 0,Y 481.648,Z 413.488,A -85,B 0,C 180,E1 -6899.418,E2 -6899.418} C_VEL
LIN {X 0,Y 481.716,Z 413.676,A -85,B 0,C 180,E1 -6901.695,E2 -6901.695} C_VEL
LIN {X 0,Y 484.624,Z 427.74,A -85,B 0,C 180,E1 -6903.944,E2 -6903.944} C_VEL
LIN {X 0,Y 484.11,Z 443.502,A -85,B 0,C 180,E1 -6906.255,E2 -6906.255} C_VEL
LIN {X 0,Y 483.436,Z 461.9,A -85,B 0,C 180,E1 -6908.912,E2 -6908.912} C_VEL
LIN {X 0,Y 482.647,Z 484.929,A -85,B 0,C 180,E1 -6912.194,E2 -6912.194} C_VEL
LIN {X 0,Y 482.352,Z 494.285,A -85,B 0,C 180,E1 -6913.498,E2 -6913.498} C_VEL
LIN {X 0,Y 484.697,Z 513.989,A -85,B 0,C 180,E1 -6913.904,E2 -6913.904} C_VEL
LIN {X 0,Y 483.83,Z 603.576,A -85,B 0,C 180,E1 -6915.354,E2 -6915.354} C_VEL
LIN {X 0,Y 483.532,Z 617.374,A -85,B 0,C 180,E1 -6915.748,E2 -6915.748} C_VEL
LIN {X 0,Y 483.087,Z 631.483,A -85,B 0,C 180,E1 -6916.325,E2 -6916.325} C_VEL
LIN {X 0,Y 482.8,Z 643.549,A -85,B 0,C 180,E1 -6917.003,E2 -6917.003} C_VEL
LIN {X 0,Y 482.396,Z 655.197,A -85,B 0,C 180,E1 -6917.856,E2 -6917.856} C_VEL
LIN {X 0,Y 482.024,Z 665.038,A -85,B 0,C 180,E1 -6918.755,E2 -6918.755} C_VEL
LIN {X 0,Y 481.681,Z 673.569,A -85,B 0,C 180,E1 -6919.704,E2 -6919.704} C_VEL
LIN {X 0,Y 481.373,Z 681.406,A -85,B 0,C 180,E1 -6920.758,E2 -6920.758} C_VEL
LIN {X 0,Y 481.172,Z 689.032,A -85,B 0,C 180,E1 -6922.024,E2 -6922.024} C_VEL
LIN {X 0,Y 481.019,Z 695.149,A -85,B 0,C 180,E1 -6923.288,E2 -6923.288} C_VEL
LIN {X 0,Y 480.963,Z 699.978,A -85,B 0,C 180,E1 -6924.55,E2 -6924.55} C_VEL
LIN {X 0,Y 480.934,Z 703.664,A -85,B 0,C 180,E1 -6925.81,E2 -6925.81} C_VEL
LIN {X 0,Y 480.979,Z 705.564,A -85,B 0,C 180,E1 -6926.649,E2 -6926.649} C_VEL
LIN {X 0,Y 480.882,Z 706.995,A -85,B 0,C 180,E1 -6927.487,E2 -6927.487} C_VEL
LIN {X 0,Y 480.849,Z 708.005,A -85,B 0,C 180,E1 -6928.325,E2 -6928.325} C_VEL
LIN {X 0,Y 480.808,Z 708.845,A -85,B 0,C 180,E1 -6930,E2 -6930} C_VEL
LIN {X 0,Y 480.813,Z 708.639,A -85,B 0,C 180,E1 -6930.838,E2 -6930.838} C_VEL
LIN {X 0,Y 480.883,Z 706.996,A -85,B 0,C 180,E1 -6932.513,E2 -6932.513} C_VEL
LIN {X 0,Y 480.992,Z 705.566,A -85,B 0,C 180,E1 -6933.351,E2 -6933.351} C_VEL
LIN {X 0,Y 480.899,Z 702.578,A -85,B 0,C 180,E1 -6934.61,E2 -6934.61} C_VEL
LIN {X 0,Y 480.987,Z 698.525,A -85,B 0,C 180,E1 -6935.871,E2 -6935.871} C_VEL
LIN {X 0,Y 481.108,Z 692.267,A -85,B 0,C 180,E1 -6937.344,E2 -6937.344} C_VEL
LIN {X 0,Y 481.307,Z 685.437,A -85,B 0,C 180,E1 -6938.608,E2 -6938.608} C_VEL
LIN {X 0,Y 481.516,Z 678.441,A -85,B 0,C 180,E1 -6939.663,E2 -6939.663} C_VEL
LIN {X 0,Y 481.793,Z 669.981,A -85,B 0,C 180,E1 -6940.719,E2 -6940.719} C_VEL
LIN {X 0,Y 482.185,Z 659.497,A -85,B 0,C 180,E1 -6941.774,E2 -6941.774} C_VEL
LIN {X 0,Y 482.534,Z 649.091,A -85,B 0,C 180,E1 -6942.619,E2 -6942.619} C_VEL
LIN {X 0,Y 482.949,Z 637.584,A -85,B 0,C 180,E1 -6943.357,E2 -6943.357} C_VEL
LIN {X 0,Y 483.291,Z 625.585,A -85,B 0,C 180,E1 -6943.937,E2 -6943.937} C_VEL
LIN {X 0,Y 483.614,Z 612.53,A -85,B 0,C 180,E1 -6944.384,E2 -6944.384} C_VEL
LIN {X 0,Y 483.861,Z 597.024,A -85,B 0,C 180,E1 -6944.698,E2 -6944.698} C_VEL
LIN {X 0,Y 484.628,Z 512.438,A -85,B 0,C 180,E1 -6946.083,E2 -6946.083} C_VEL
LIN {X 0,Y 482.194,Z 491.482,A -85,B 0,C 180,E1 -6946.54,E2 -6946.54} C_VEL
LIN {X 0,Y 482.869,Z 468.459,A -85,B 0,C 180,E1 -6949.779,E2 -6949.779} C_VEL
LIN {X 0,Y 483.463,Z 448.401,A -85,B 0,C 180,E1 -6952.658,E2 -6952.658} C_VEL
LIN {X 0,Y 484.258,Z 426.972,A -85,B 0,C 180,E1 -6955.81,E2 -6955.81} C_VEL
LIN {X 0,Y 482.83,Z 418.621,A -85,B 0,C 180,E1 -6957.167,E2 -6957.167} C_VEL
LIN {X 0,Y 481.669,Z 413.49,A -85,B 0,C 180,E1 -6958.071,E2 -6958.071} C_VEL
LIN {X 0,Y 481.643,Z 413.492,A -85,B 0,C 180,E1 -6960.711,E2 -6960.711} C_VEL
LIN {X 0,Y 481.699,Z 413.486,A -85,B 0,C 180,E1 -6963.733,E2 -6963.733} C_VEL
LIN {X 0,Y 481.622,Z 413.491,A -85,B 0,C 180,E1 -6966.747,E2 -6966.747} C_VEL
LIN {X 0,Y 481.67,Z 413.486,A -85,B 0,C 180,E1 -6969.941,E2 -6969.941} C_VEL
LIN {X 0,Y 481.63,Z 413.494,A -85,B 0,C 180,E1 -6973.147,E2 -6973.147} C_VEL
LIN {X 0,Y 481.661,Z 413.488,A -85,B 0,C 180,E1 -6975.641,E2 -6975.641} C_VEL
LIN {X 0,Y 481.658,Z 413.489,A -85,B 0,C 180,E1 -6978.958,E2 -6978.958} C_VEL
LIN {X 0,Y 481.657,Z 413.485,A -85,B 0,C 180,E1 -6981.993,E2 -6981.993} C_VEL
LIN {X 0,Y 481.692,Z 413.483,A -85,B 0,C 180,E1 -6985.318,E2 -6985.318} C_VEL
LIN {X 0,Y 481.648,Z 413.488,A -85,B 0,C 180,E1 -6988.312,E2 -6988.312} C_VEL
LIN {X 0,Y 481.701,Z 413.484,A -85,B 0,C 180,E1 -6991.219,E2 -6991.219} C_VEL
LIN {X 0,Y 481.692,Z 413.483,A -85,B 0,C 180,E1 -6994.042,E2 -6994.042} C_VEL
LIN {X 0,Y 481.677,Z 413.49,A -85,B 0,C 180,E1 -6996.812,E2 -6996.812} C_VEL
LIN {X 0,Y 481.698,Z 413.482,A -85,B 0,C 180,E1 -6999.503,E2 -6999.503} C_VEL
LIN {X 0,Y 481.69,Z 413.487,A -85,B 0,C 180,E1 -7002.158,E2 -7002.158} C_VEL
LIN {X 0,Y 481.71,Z 413.604,A -85,B 0,C 180,E1 -7003.613,E2 -7003.613} C_VEL
LIN {X 0,Y 485.077,Z 423.17,A -85,B 0,C 180,E1 -7003.913,E2 -7003.913} C_VEL
LIN {X 0,Y 484.065,Z 515.91,A -85,B 0,C 180,E1 -7005.496,E2 -7005.496} C_VEL
LIN {X 0,Y 483.878,Z 529.285,A -85,B 0,C 180,E1 -7005.893,E2 -7005.893} C_VEL
LIN {X 0,Y 483.614,Z 542.001,A -85,B 0,C 180,E1 -7006.448,E2 -7006.448} C_VEL
LIN {X 0,Y 483.297,Z 553.897,A -85,B 0,C 180,E1 -7007.151,E2 -7007.151} C_VEL
LIN {X 0,Y 482.927,Z 565.534,A -85,B 0,C 180,E1 -7008.031,E2 -7008.031} C_VEL
LIN {X 0,Y 482.629,Z 574.488,A -85,B 0,C 180,E1 -7008.875,E2 -7008.875} C_VEL
LIN {X 0,Y 482.255,Z 583.641,A -85,B 0,C 180,E1 -7009.928,E2 -7009.928} C_VEL
LIN {X 0,Y 481.892,Z 592.502,A -85,B 0,C 180,E1 -7011.191,E2 -7011.191} C_VEL
LIN {X 0,Y 481.623,Z 599.592,A -85,B 0,C 180,E1 -7012.454,E2 -7012.454} C_VEL
LIN {X 0,Y 481.467,Z 605.193,A -85,B 0,C 180,E1 -7013.715,E2 -7013.715} C_VEL
LIN {X 0,Y 481.23,Z 609.584,A -85,B 0,C 180,E1 -7014.973,E2 -7014.973} C_VEL
LIN {X 0,Y 481.261,Z 611.872,A -85,B 0,C 180,E1 -7015.813,E2 -7015.813} C_VEL
LIN {X 0,Y 481.116,Z 613.748,A -85,B 0,C 180,E1 -7016.65,E2 -7016.65} C_VEL
LIN {X 0,Y 480.985,Z 615.18,A -85,B 0,C 180,E1 -7017.488,E2 -7017.488} C_VEL
LIN {X 0,Y 480.886,Z 616.756,A -85,B 0,C 180,E1 -7019.163,E2 -7019.163} C_VEL
LIN {X 0,Y 480.878,Z 616.958,A -85,B 0,C 180,E1 -7020,E2 -7020} C_VEL
LIN {X 0,Y 480.88,Z 616.731,A -85,B 0,C 180,E1 -7020.837,E2 -7020.837} C_VEL
LIN {X 0,Y 480.968,Z 615.064,A -85,B 0,C 180,E1 -7022.513,E2 -7022.513} C_VEL
LIN {X 0,Y 481.114,Z 613.626,A -85,B 0,C 180,E1 -7023.35,E2 -7023.35} C_VEL
LIN {X 0,Y 481.222,Z 610.64,A -85,B 0,C 180,E1 -7024.607,E2 -7024.607} C_VEL
LIN {X 0,Y 481.222,Z 606.617,A -85,B 0,C 180,E1 -7025.868,E2 -7025.868} C_VEL
LIN {X 0,Y 481.454,Z 600.848,A -85,B 0,C 180,E1 -7027.244,E2 -7027.244} C_VEL
LIN {X 0,Y 481.74,Z 593.599,A -85,B 0,C 180,E1 -7028.6,E2 -7028.6} C_VEL
LIN {X 0,Y 482.039,Z 585.141,A -85,B 0,C 180,E1 -7029.864,E2 -7029.864} C_VEL
LIN {X 0,Y 482.417,Z 576.399,A -85,B 0,C 180,E1 -7030.917,E2 -7030.917} C_VEL
LIN {X 0,Y 482.794,Z 565.628,A -85,B 0,C 180,E1 -7031.972,E2 -7031.972} C_VEL
LIN {X 0,Y 483.175,Z 554.891,A -85,B 0,C 180,E1 -7032.814,E2 -7032.814} C_VEL
LIN {X 0,Y 483.469,Z 542.802,A -85,B 0,C 180,E1 -7033.557,E2 -7033.557} C_VEL
LIN {X 0,Y 483.765,Z 530.247,A -85,B 0,C 180,E1 -7034.137,E2 -7034.137} C_VEL
LIN {X 0,Y 484.035,Z 517.036,A -85,B 0,C 180,E1 -7034.559,E2 -7034.559} C_VEL
LIN {X 0,Y 484.222,Z 499.931,A -85,B 0,C 180,E1 -7034.875,E2 -7034.875} C_VEL
LIN {X 0,Y 484.786,Z 422.72,A -85,B 0,C 180,E1 -7036.127,E2 -7036.127} C_VEL
LIN {X 0,Y 481.691,Z 413.483,A -85,B 0,C 180,E1 -7036.396,E2 -7036.396} C_VEL
LIN {X 0,Y 481.703,Z 413.488,A -85,B 0,C 180,E1 -7039.607,E2 -7039.607} C_VEL
LIN {X 0,Y 481.651,Z 413.484,A -85,B 0,C 180,E1 -7042.295,E2 -7042.295} C_VEL
LIN {X 0,Y 481.675,Z 413.487,A -85,B 0,C 180,E1 -7045.227,E2 -7045.227} C_VEL
LIN {X 0,Y 481.694,Z 413.478,A -85,B 0,C 180,E1 -7047.832,E2 -7047.832} C_VEL
LIN {X 0,Y 481.649,Z 413.487,A -85,B 0,C 180,E1 -7050.711,E2 -7050.711} C_VEL
LIN {X 0,Y 481.7,Z 413.47,A -85,B 0,C 180,E1 -7053.733,E2 -7053.733} C_VEL
LIN {X 0,Y 481.629,Z 413.492,A -85,B 0,C 180,E1 -7056.747,E2 -7056.747} C_VEL
LIN {X 0,Y 481.68,Z 413.475,A -85,B 0,C 180,E1 -7059.94,E2 -7059.94} C_VEL
LIN {X 0,Y 481.642,Z 413.49,A -85,B 0,C 180,E1 -7063.3,E2 -7063.3} C_VEL
LIN {X 0,Y 481.661,Z 413.477,A -85,B 0,C 180,E1 -7065.641,E2 -7065.641} C_VEL
LIN {X 0,Y 481.659,Z 413.485,A -85,B 0,C 180,E1 -7068.958,E2 -7068.958} C_VEL
LIN {X 0,Y 481.653,Z 413.487,A -85,B 0,C 180,E1 -7071.993,E2 -7071.993} C_VEL
LIN {X 0,Y 481.635,Z 413.49,A -85,B 0,C 180,E1 -7074.307,E2 -7074.307} C_VEL
LIN {X 0,Y 480.996,Z 413.57,A -85,B 0,C 180,E1 -7075.005,E2 -7075.005} C_VEL
LIN {X 0,Y 478.181,Z 413.92,A -85,B 0,C 180,E1 -7076.14,E2 -7076.14} C_VEL
LIN {X 0,Y 475.773,Z 414.22,A -85,B 0,C 180,E1 -7077.055,E2 -7077.055} C_VEL
LIN {X 0,Y 474.716,Z 414.351,A -85,B 0,C 180,E1 -7077.761,E2 -7077.761} C_VEL
LIN {X 0,Y 474.618,Z 414.363,A -85,B 0,C 180,E1 -7078,E2 -7078} C_VEL
LIN {X 0,Y 474.601,Z 414.37,A -85,B 0,C 180,E1 -7080.89,E2 -7080.89} C_VEL
LIN {X 0,Y 474.652,Z 414.471,A -85,B 0,C 180,E1 -7084.198,E2 -7084.198} C_VEL
LIN {X 0,Y 476.883,Z 425.985,A -85,B 0,C 180,E1 -7086.197,E2 -7086.197} C_VEL
LIN {X 0,Y 476.592,Z 439.219,A -85,B 0,C 180,E1 -7088.367,E2 -7088.367} C_VEL
LIN {X 0,Y 475.979,Z 458.669,A -85,B 0,C 180,E1 -7091.491,E2 -7091.491} C_VEL
LIN {X 0,Y 475.726,Z 470.565,A -85,B 0,C 180,E1 -7093.299,E2 -7093.299} C_VEL
LIN {X 0,Y 478.13,Z 485.496,A -85,B 0,C 180,E1 -7093.617,E2 -7093.617} C_VEL
LIN {X 0,Y 477.442,Z 578.867,A -85,B 0,C 180,E1 -7095.045,E2 -7095.045} C_VEL
LIN {X 0,Y 477.207,Z 591.826,A -85,B 0,C 180,E1 -7095.392,E2 -7095.392} C_VEL
LIN {X 0,Y 476.846,Z 603.787,A -85,B 0,C 180,E1 -7095.871,E2 -7095.871} C_VEL
LIN {X 0,Y 476.499,Z 614.652,A -85,B 0,C 180,E1 -7096.46,E2 -7096.46} C_VEL
LIN {X 0,Y 476.116,Z 625.443,A -85,B 0,C 180,E1 -7097.208,E2 -7097.208} C_VEL
LIN {X 0,Y 475.621,Z 636.513,A -85,B 0,C 180,E1 -7098.169,E2 -7098.169} C_VEL
LIN {X 0,Y 475.143,Z 645.486,A -85,B 0,C 180,E1 -7099.129,E2 -7099.129} C_VEL
LIN {X 0,Y 474.709,Z 655.128,A -85,B 0,C 180,E1 -7100.412,E2 -7100.412} C_VEL
LIN {X 0,Y 474.36,Z 662.882,A -85,B 0,C 180,E1 -7101.694,E2 -7101.694} C_VEL
LIN {X 0,Y 474.147,Z 668.124,A -85,B 0,C 180,E1 -7102.762,E2 -7102.762} C_VEL
LIN {X 0,Y 474.077,Z 673.244,A -85,B 0,C 180,E1 -7104.044,E2 -7104.044} C_VEL
LIN {X 0,Y 473.82,Z 677.217,A -85,B 0,C 180,E1 -7105.321,E2 -7105.321} C_VEL
LIN {X 0,Y 473.839,Z 680.143,A -85,B 0,C 180,E1 -7106.599,E2 -7106.599} C_VEL
LIN {X 0,Y 473.763,Z 681.568,A -85,B 0,C 180,E1 -7107.449,E2 -7107.449} C_VEL
LIN {X 0,Y 473.689,Z 683.181,A -85,B 0,C 180,E1 -7109.15,E2 -7109.15} C_VEL
LIN {X 0,Y 473.67,Z 683.419,A -85,B 0,C 180,E1 -7110,E2 -7110} C_VEL
LIN {X 0,Y 473.689,Z 683.231,A -85,B 0,C 180,E1 -7110.85,E2 -7110.85} C_VEL
LIN {X 0,Y 473.763,Z 681.683,A -85,B 0,C 180,E1 -7112.551,E2 -7112.551} C_VEL
LIN {X 0,Y 473.839,Z 680.322,A -85,B 0,C 180,E1 -7113.401,E2 -7113.401} C_VEL
LIN {X 0,Y 473.819,Z 677.462,A -85,B 0,C 180,E1 -7114.679,E2 -7114.679} C_VEL
LIN {X 0,Y 474.042,Z 673.57,A -85,B 0,C 180,E1 -7115.957,E2 -7115.957} C_VEL
LIN {X 0,Y 474.146,Z 668.534,A -85,B 0,C 180,E1 -7117.238,E2 -7117.238} C_VEL
LIN {X 0,Y 474.417,Z 662.181,A -85,B 0,C 180,E1 -7118.519,E2 -7118.519} C_VEL
LIN {X 0,Y 474.746,Z 654.29,A -85,B 0,C 180,E1 -7119.802,E2 -7119.802} C_VEL
LIN {X 0,Y 475.099,Z 646.23,A -85,B 0,C 180,E1 -7120.872,E2 -7120.872} C_VEL
LIN {X 0,Y 475.647,Z 636.334,A -85,B 0,C 180,E1 -7121.938,E2 -7121.938} C_VEL
LIN {X 0,Y 476.122,Z 624.829,A -85,B 0,C 180,E1 -7122.931,E2 -7122.931} C_VEL
LIN {X 0,Y 476.512,Z 614.355,A -85,B 0,C 180,E1 -7123.65,E2 -7123.65} C_VEL
LIN {X 0,Y 476.892,Z 603.404,A -85,B 0,C 180,E1 -7124.237,E2 -7124.237} C_VEL
LIN {X 0,Y 477.229,Z 590.444,A -85,B 0,C 180,E1 -7124.744,E2 -7124.744} C_VEL
LIN {X 0,Y 477.506,Z 578,A -85,B 0,C 180,E1 -7125.062,E2 -7125.062} C_VEL
LIN {X 0,Y 478.143,Z 484.938,A -85,B 0,C 180,E1 -7126.482,E2 -7126.482} C_VEL
LIN {X 0,Y 475.727,Z 470.525,A -85,B 0,C 180,E1 -7126.796,E2 -7126.796} C_VEL
LIN {X 0,Y 476.136,Z 453.625,A -85,B 0,C 180,E1 -7129.406,E2 -7129.406} C_VEL
LIN {X 0,Y 476.687,Z 435.835,A -85,B 0,C 180,E1 -7132.289,E2 -7132.289} C_VEL
LIN {X 0,Y 476.94,Z 426.48,A -85,B 0,C 180,E1 -7133.818,E2 -7133.818} C_VEL
LIN {X 0,Y 474.633,Z 414.368,A -85,B 0,C 180,E1 -7135.93,E2 -7135.93} C_VEL
LIN {X 0,Y 474.603,Z 414.368,A -85,B 0,C 180,E1 -7139.253,E2 -7139.253} C_VEL
LIN {X 0,Y 474.618,Z 414.364,A -85,B 0,C 180,E1 -7142.43,E2 -7142.43} C_VEL
LIN {X 0,Y 474.614,Z 414.369,A -85,B 0,C 180,E1 -7145.469,E2 -7145.469} C_VEL
LIN {X 0,Y 474.613,Z 414.362,A -85,B 0,C 180,E1 -7148.457,E2 -7148.457} C_VEL
LIN {X 0,Y 474.623,Z 414.363,A -85,B 0,C 180,E1 -7151.785,E2 -7151.785} C_VEL
LIN {X 0,Y 474.624,Z 414.361,A -85,B 0,C 180,E1 -7154.703,E2 -7154.703} C_VEL
LIN {X 0,Y 474.628,Z 414.356,A -85,B 0,C 180,E1 -7157.763,E2 -7157.763} C_VEL
LIN {X 0,Y 474.648,Z 414.361,A -85,B 0,C 180,E1 -7160.454,E2 -7160.454} C_VEL
LIN {X 0,Y 474.587,Z 414.357,A -85,B 0,C 180,E1 -7163.676,E2 -7163.676} C_VEL
LIN {X 0,Y 474.646,Z 414.364,A -85,B 0,C 180,E1 -7166.78,E2 -7166.78} C_VEL
LIN {X 0,Y 474.6,Z 414.365,A -85,B 0,C 180,E1 -7169.769,E2 -7169.769} C_VEL
LIN {X 0,Y 474.639,Z 414.363,A -85,B 0,C 180,E1 -7172.676,E2 -7172.676} C_VEL
LIN {X 0,Y 474.632,Z 414.428,A -85,B 0,C 180,E1 -7174.197,E2 -7174.197} C_VEL
LIN {X 0,Y 476.884,Z 426.161,A -85,B 0,C 180,E1 -7176.199,E2 -7176.199} C_VEL
LIN {X 0,Y 476.736,Z 437.123,A -85,B 0,C 180,E1 -7177.964,E2 -7177.964} C_VEL
LIN {X 0,Y 476.139,Z 457.903,A -85,B 0,C 180,E1 -7181.274,E2 -7181.274} C_VEL
LIN {X 0,Y 475.742,Z 471.043,A -85,B 0,C 180,E1 -7183.353,E2 -7183.353} C_VEL
LIN {X 0,Y 477.949,Z 485.182,A -85,B 0,C 180,E1 -7183.671,E2 -7183.671} C_VEL
LIN {X 0,Y 477.079,Z 580.285,A -85,B 0,C 180,E1 -7185.251,E2 -7185.251} C_VEL
LIN {X 0,Y 476.724,Z 593.796,A -85,B 0,C 180,E1 -7185.649,E2 -7185.649} C_VEL
LIN {X 0,Y 476.435,Z 606.17,A -85,B 0,C 180,E1 -7186.185,E2 -7186.185} C_VEL
LIN {X 0,Y 475.987,Z 618.447,A -85,B 0,C 180,E1 -7186.903,E2 -7186.903} C_VEL
LIN {X 0,Y 475.692,Z 629.621,A -85,B 0,C 180,E1 -7187.743,E2 -7187.743} C_VEL
LIN {X 0,Y 475.22,Z 639.844,A -85,B 0,C 180,E1 -7188.699,E2 -7188.699} C_VEL
LIN {X 0,Y 474.872,Z 649.133,A -85,B 0,C 180,E1 -7189.77,E2 -7189.77} C_VEL
LIN {X 0,Y 474.513,Z 656.783,A -85,B 0,C 180,E1 -7190.838,E2 -7190.838} C_VEL
LIN {X 0,Y 474.218,Z 664.272,A -85,B 0,C 180,E1 -7192.121,E2 -7192.121} C_VEL
LIN {X 0,Y 474.008,Z 671.354,A -85,B 0,C 180,E1 -7193.671,E2 -7193.671} C_VEL
LIN {X 0,Y 473.854,Z 675.658,A -85,B 0,C 180,E1 -7194.894,E2 -7194.894} C_VEL
LIN {X 0,Y 473.835,Z 678.03,A -85,B 0,C 180,E1 -7195.747,E2 -7195.747} C_VEL
LIN {X 0,Y 473.837,Z 679.954,A -85,B 0,C 180,E1 -7196.599,E2 -7196.599} C_VEL
LIN {X 0,Y 473.763,Z 681.466,A -85,B 0,C 180,E1 -7197.449,E2 -7197.449} C_VEL
LIN {X 0,Y 473.727,Z 682.512,A -85,B 0,C 180,E1 -7198.3,E2 -7198.3} C_VEL
LIN {X 0,Y 473.67,Z 683.422,A -85,B 0,C 180,E1 -7200,E2 -7200} C_VEL
LIN {X 0,Y 473.689,Z 683.235,A -85,B 0,C 180,E1 -7200.85,E2 -7200.85} C_VEL
LIN {X 0,Y 473.727,Z 682.642,A -85,B 0,C 180,E1 -7201.7,E2 -7201.7} C_VEL
LIN {X 0,Y 473.763,Z 681.658,A -85,B 0,C 180,E1 -7202.551,E2 -7202.551} C_VEL
LIN {X 0,Y 473.836,Z 680.224,A -85,B 0,C 180,E1 -7203.401,E2 -7203.401} C_VEL
LIN {X 0,Y 473.806,Z 677.256,A -85,B 0,C 180,E1 -7204.679,E2 -7204.679} C_VEL
LIN {X 0,Y 474.014,Z 673.206,A -85,B 0,C 180,E1 -7205.957,E2 -7205.957} C_VEL
LIN {X 0,Y 474.129,Z 666.997,A -85,B 0,C 180,E1 -7207.452,E2 -7207.452} C_VEL
LIN {X 0,Y 474.411,Z 660.134,A -85,B 0,C 180,E1 -7208.734,E2 -7208.734} C_VEL
LIN {X 0,Y 474.74,Z 651.571,A -85,B 0,C 180,E1 -7210.017,E2 -7210.017} C_VEL
LIN {X 0,Y 475.126,Z 641.756,A -85,B 0,C 180,E1 -7211.195,E2 -7211.195} C_VEL
LIN {X 0,Y 475.626,Z 630.824,A -85,B 0,C 180,E1 -7212.246,E2 -7212.246} C_VEL
LIN {X 0,Y 475.973,Z 619.462,A -85,B 0,C 180,E1 -7213.111,E2 -7213.111} C_VEL
LIN {X 0,Y 476.315,Z 607.622,A -85,B 0,C 180,E1 -7213.818,E2 -7213.818} C_VEL
LIN {X 0,Y 476.733,Z 594.975,A -85,B 0,C 180,E1 -7214.378,E2 -7214.378} C_VEL
LIN {X 0,Y 477.003,Z 581.881,A -85,B 0,C 180,E1 -7214.778,E2 -7214.778} C_VEL
LIN {X 0,Y 478.099,Z 484.742,A -85,B 0,C 180,E1 -7216.46,E2 -7216.46} C_VEL
LIN {X 0,Y 475.897,Z 471.535,A -85,B 0,C 180,E1 -7216.806,E2 -7216.806} C_VEL
LIN {X 0,Y 476.369,Z 452.084,A -85,B 0,C 180,E1 -7219.836,E2 -7219.836} C_VEL
LIN {X 0,Y 476.848,Z 433.003,A -85,B 0,C 180,E1 -7222.761,E2 -7222.761} C_VEL
LIN {X 0,Y 476.816,Z 425.247,A -85,B 0,C 180,E1 -7223.957,E2 -7223.957} C_VEL
LIN {X 0,Y 474.621,Z 414.368,A -85,B 0,C 180,E1 -7225.772,E2 -7225.772} C_VEL
LIN {X 0,Y 474.601,Z 414.37,A -85,B 0,C 180,E1 -7229.11,E2 -7229.11} C_VEL
LIN {X 0,Y 474.617,Z 414.364,A -85,B 0,C 180,E1 -7232.43,E2 -7232.43} C_VEL
LIN {X 0,Y 474.614,Z 414.368,A -85,B 0,C 180,E1 -7235.469,E2 -7235.469} C_VEL
LIN {X 0,Y 474.612,Z 414.363,A -85,B 0,C 180,E1 -7238.457,E2 -7238.457} C_VEL
LIN {X 0,Y 474.63,Z 414.365,A -85,B 0,C 180,E1 -7240.959,E2 -7240.959} C_VEL
LIN {X 0,Y 474.612,Z 414.363,A -85,B 0,C 180,E1 -7244.105,E2 -7244.105} C_VEL
LIN {X 0,Y 474.618,Z 414.365,A -85,B 0,C 180,E1 -7247.066,E2 -7247.066} C_VEL
LIN {X 0,Y 474.647,Z 414.362,A -85,B 0,C 180,E1 -7250.454,E2 -7250.454} C_VEL
LIN {X 0,Y 474.586,Z 414.366,A -85,B 0,C 180,E1 -7253.676,E2 -7253.676} C_VEL
LIN {X 0,Y 474.645,Z 414.364,A -85,B 0,C 180,E1 -7256.78,E2 -7256.78} C_VEL
LIN {X 0,Y 474.599,Z 414.367,A -85,B 0,C 180,E1 -7259.769,E2 -7259.769} C_VEL
LIN {X 0,Y 474.662,Z 414.554,A -85,B 0,C 180,E1 -7261.477,E2 -7261.477} C_VEL
LIN {X 0,Y 477.692,Z 429.001,A -85,B 0,C 180,E1 -7263.826,E2 -7263.826} C_VEL
LIN {X 0,Y 477.297,Z 443.05,A -85,B 0,C 180,E1 -7265.913,E2 -7265.913} C_VEL
LIN {X 0,Y 476.466,Z 462.853,A -85,B 0,C 180,E1 -7268.815,E2 -7268.815} C_VEL
LIN {X 0,Y 475.624,Z 485.859,A -85,B 0,C 180,E1 -7272.145,E2 -7272.145} C_VEL
LIN {X 0,Y 475.363,Z 493.521,A -85,B 0,C 180,E1 -7273.245,E2 -7273.245} C_VEL
LIN {X 0,Y 477.844,Z 513.843,A -85,B 0,C 180,E1 -7273.682,E2 -7273.682} C_VEL
LIN {X 0,Y 476.922,Z 603.141,A -85,B 0,C 180,E1 -7275.165,E2 -7275.165} C_VEL
LIN {X 0,Y 476.58,Z 619.207,A -85,B 0,C 180,E1 -7275.618,E2 -7275.618} C_VEL
LIN {X 0,Y 476.162,Z 632.455,A -85,B 0,C 180,E1 -7276.177,E2 -7276.177} C_VEL
LIN {X 0,Y 475.815,Z 644.335,A -85,B 0,C 180,E1 -7276.874,E2 -7276.874} C_VEL
LIN {X 0,Y 475.397,Z 655.57,A -85,B 0,C 180,E1 -7277.72,E2 -7277.72} C_VEL
LIN {X 0,Y 474.989,Z 665.914,A -85,B 0,C 180,E1 -7278.694,E2 -7278.694} C_VEL
LIN {X 0,Y 474.568,Z 675.061,A -85,B 0,C 180,E1 -7279.763,E2 -7279.763} C_VEL
LIN {X 0,Y 474.253,Z 683.947,A -85,B 0,C 180,E1 -7281.048,E2 -7281.048} C_VEL
LIN {X 0,Y 474.037,Z 691.066,A -85,B 0,C 180,E1 -7282.332,E2 -7282.332} C_VEL
LIN {X 0,Y 473.889,Z 696.428,A -85,B 0,C 180,E1 -7283.537,E2 -7283.537} C_VEL
LIN {X 0,Y 473.842,Z 701.146,A -85,B 0,C 180,E1 -7284.894,E2 -7284.894} C_VEL
LIN {X 0,Y 473.827,Z 703.476,A -85,B 0,C 180,E1 -7285.747,E2 -7285.747} C_VEL
LIN {X 0,Y 473.9,Z 705.376,A -85,B 0,C 180,E1 -7286.599,E2 -7286.599} C_VEL
LIN {X 0,Y 473.798,Z 706.807,A -85,B 0,C 180,E1 -7287.449,E2 -7287.449} C_VEL
LIN {X 0,Y 473.739,Z 708.433,A -85,B 0,C 180,E1 -7289.15,E2 -7289.15} C_VEL
LIN {X 0,Y 473.731,Z 708.657,A -85,B 0,C 180,E1 -7290,E2 -7290} C_VEL
LIN {X 0,Y 473.739,Z 708.453,A -85,B 0,C 180,E1 -7290.85,E2 -7290.85} C_VEL
LIN {X 0,Y 473.8,Z 706.808,A -85,B 0,C 180,E1 -7292.551,E2 -7292.551} C_VEL
LIN {X 0,Y 473.913,Z 705.378,A -85,B 0,C 180,E1 -7293.401,E2 -7293.401} C_VEL
LIN {X 0,Y 473.814,Z 702.391,A -85,B 0,C 180,E1 -7294.679,E2 -7294.679} C_VEL
LIN {X 0,Y 473.858,Z 697.513,A -85,B 0,C 180,E1 -7296.177,E2 -7296.177} C_VEL
LIN {X 0,Y 474.045,Z 691.071,A -85,B 0,C 180,E1 -7297.668,E2 -7297.668} C_VEL
LIN {X 0,Y 474.271,Z 683.954,A -85,B 0,C 180,E1 -7298.951,E2 -7298.951} C_VEL
LIN {X 0,Y 474.577,Z 675.056,A -85,B 0,C 180,E1 -7300.236,E2 -7300.236} C_VEL
LIN {X 0,Y 474.996,Z 665.903,A -85,B 0,C 180,E1 -7301.306,E2 -7301.306} C_VEL
LIN {X 0,Y 475.41,Z 655.737,A -85,B 0,C 180,E1 -7302.266,E2 -7302.266} C_VEL
LIN {X 0,Y 475.78,Z 644.329,A -85,B 0,C 180,E1 -7303.127,E2 -7303.127} C_VEL
LIN {X 0,Y 476.196,Z 632.444,A -85,B 0,C 180,E1 -7303.822,E2 -7303.822} C_VEL
LIN {X 0,Y 476.574,Z 619.946,A -85,B 0,C 180,E1 -7304.355,E2 -7304.355} C_VEL
LIN {X 0,Y 476.844,Z 607.025,A -85,B 0,C 180,E1 -7304.729,E2 -7304.729} C_VEL
LIN {X 0,Y 477.73,Z 519.06,A -85,B 0,C 180,E1 -7306.201,E2 -7306.201} C_VEL
LIN {X 0,Y 477.619,Z 511.678,A -85,B 0,C 180,E1 -7306.337,E2 -7306.337} C_VEL
LIN {X 0,Y 475.189,Z 490.485,A -85,B 0,C 180,E1 -7306.831,E2 -7306.831} C_VEL
LIN {X 0,Y 475.86,Z 467.841,A -85,B 0,C 180,E1 -7310.083,E2 -7310.083} C_VEL
LIN {X 0,Y 476.516,Z 449.408,A -85,B 0,C 180,E1 -7312.778,E2 -7312.778} C_VEL
LIN {X 0,Y 477.398,Z 428.393,A -85,B 0,C 180,E1 -7315.934,E2 -7315.934} C_VEL
LIN {X 0,Y 475.258,Z 417.168,A -85,B 0,C 180,E1 -7317.825,E2 -7317.825} C_VEL
LIN {X 0,Y 474.635,Z 414.366,A -85,B 0,C 180,E1 -7318.344,E2 -7318.344} C_VEL
LIN {X 0,Y 474.599,Z 414.372,A -85,B 0,C 180,E1 -7321.218,E2 -7321.218} C_VEL
LIN {X 0,Y 474.633,Z 414.362,A -85,B 0,C 180,E1 -7324.241,E2 -7324.241} C_VEL
LIN {X 0,Y 474.587,Z 414.371,A -85,B 0,C 180,E1 -7327.384,E2 -7327.384} C_VEL
LIN {X 0,Y 474.616,Z 414.364,A -85,B 0,C 180,E1 -7330.658,E2 -7330.658} C_VEL
LIN {X 0,Y 474.595,Z 414.369,A -85,B 0,C 180,E1 -7333.48,E2 -7333.48} C_VEL
LIN {X 0,Y 474.604,Z 414.365,A -85,B 0,C 180,E1 -7336.519,E2 -7336.519} C_VEL
LIN {X 0,Y 474.619,Z 414.366,A -85,B 0,C 180,E1 -7339.342,E2 -7339.342} C_VEL
LIN {X 0,Y 474.612,Z 414.364,A -85,B 0,C 180,E1 -7341.704,E2 -7341.704} C_VEL
LIN {X 0,Y 474.628,Z 414.363,A -85,B 0,C 180,E1 -7344.726,E2 -7344.726} C_VEL
LIN {X 0,Y 474.638,Z 414.36,A -85,B 0,C 180,E1 -7347.788,E2 -7347.788} C_VEL
LIN {X 0,Y 474.626,Z 414.367,A -85,B 0,C 180,E1 -7350.885,E2 -7350.885} C_VEL
LIN {X 0,Y 474.656,Z 414.359,A -85,B 0,C 180,E1 -7353.628,E2 -7353.628} C_VEL
LIN {X 0,Y 474.638,Z 414.368,A -85,B 0,C 180,E1 -7356.642,E2 -7356.642} C_VEL
LIN {X 0,Y 474.656,Z 414.361,A -85,B 0,C 180,E1 -7360.09,E2 -7360.09} C_VEL
LIN {X 0,Y 474.651,Z 414.362,A -85,B 0,C 180,E1 -7363.326,E2 -7363.326} C_VEL
LIN {X 0,Y 478.328,Z 424.75,A -85,B 0,C 180,E1 -7363.68,E2 -7363.68} C_VEL
LIN {X 0,Y 477.192,Z 517.52,A -85,B 0,C 180,E1 -7365.31,E2 -7365.31} C_VEL
LIN {X 0,Y 477.012,Z 530.596,A -85,B 0,C 180,E1 -7365.713,E2 -7365.713} C_VEL
LIN {X 0,Y 476.767,Z 542.63,A -85,B 0,C 180,E1 -7366.249,E2 -7366.249} C_VEL
LIN {X 0,Y 476.417,Z 554.531,A -85,B 0,C 180,E1 -7366.962,E2 -7366.962} C_VEL
LIN {X 0,Y 476.012,Z 566.154,A -85,B 0,C 180,E1 -7367.855,E2 -7367.855} C_VEL
LIN {X 0,Y 475.697,Z 575.109,A -85,B 0,C 180,E1 -7368.711,E2 -7368.711} C_VEL
LIN {X 0,Y 475.302,Z 584.269,A -85,B 0,C 180,E1 -7369.78,E2 -7369.78} C_VEL
LIN {X 0,Y 474.926,Z 593.135,A -85,B 0,C 180,E1 -7371.061,E2 -7371.061} C_VEL
LIN {X 0,Y 474.611,Z 600.254,A -85,B 0,C 180,E1 -7372.341,E2 -7372.341} C_VEL
LIN {X 0,Y 474.449,Z 605.872,A -85,B 0,C 180,E1 -7373.621,E2 -7373.621} C_VEL
LIN {X 0,Y 474.201,Z 610.273,A -85,B 0,C 180,E1 -7374.898,E2 -7374.898} C_VEL
LIN {X 0,Y 474.23,Z 612.564,A -85,B 0,C 180,E1 -7375.751,E2 -7375.751} C_VEL
LIN {X 0,Y 474.073,Z 614.442,A -85,B 0,C 180,E1 -7376.6,E2 -7376.6} C_VEL
LIN {X 0,Y 473.927,Z 615.874,A -85,B 0,C 180,E1 -7377.45,E2 -7377.45} C_VEL
LIN {X 0,Y 473.821,Z 617.443,A -85,B 0,C 180,E1 -7379.15,E2 -7379.15} C_VEL
LIN {X 0,Y 473.811,Z 617.638,A -85,B 0,C 180,E1 -7380,E2 -7380} C_VEL
LIN {X 0,Y 473.813,Z 617.4,A -85,B 0,C 180,E1 -7380.85,E2 -7380.85} C_VEL
LIN {X 0,Y 473.911,Z 615.707,A -85,B 0,C 180,E1 -7382.55,E2 -7382.55} C_VEL
LIN {X 0,Y 474.071,Z 614.251,A -85,B 0,C 180,E1 -7383.4,E2 -7383.4} C_VEL
LIN {X 0,Y 474.162,Z 611.239,A -85,B 0,C 180,E1 -7384.676,E2 -7384.676} C_VEL
LIN {X 0,Y 474.184,Z 607.18,A -85,B 0,C 180,E1 -7385.955,E2 -7385.955} C_VEL
LIN {X 0,Y 474.43,Z 601.013,A -85,B 0,C 180,E1 -7387.426,E2 -7387.426} C_VEL
LIN {X 0,Y 474.735,Z 594.068,A -85,B 0,C 180,E1 -7388.728,E2 -7388.728} C_VEL
LIN {X 0,Y 475.072,Z 585.538,A -85,B 0,C 180,E1 -7390.01,E2 -7390.01} C_VEL
LIN {X 0,Y 475.446,Z 576.736,A -85,B 0,C 180,E1 -7391.079,E2 -7391.079} C_VEL
LIN {X 0,Y 475.862,Z 565.888,A -85,B 0,C 180,E1 -7392.149,E2 -7392.149} C_VEL
LIN {X 0,Y 476.275,Z 554.492,A -85,B 0,C 180,E1 -7393.04,E2 -7393.04} C_VEL
LIN {X 0,Y 476.576,Z 542.814,A -85,B 0,C 180,E1 -7393.756,E2 -7393.756} C_VEL
LIN {X 0,Y 476.884,Z 530.084,A -85,B 0,C 180,E1 -7394.346,E2 -7394.346} C_VEL
LIN {X 0,Y 477.145,Z 517.475,A -85,B 0,C 180,E1 -7394.746,E2 -7394.746} C_VEL
LIN {X 0,Y 477.311,Z 502.034,A -85,B 0,C 180,E1 -7395.041,E2 -7395.041} C_VEL
LIN {X 0,Y 477.938,Z 424.198,A -85,B 0,C 180,E1 -7396.333,E2 -7396.333} C_VEL
LIN {X 0,Y 474.642,Z 414.362,A -85,B 0,C 180,E1 -7396.63,E2 -7396.63} C_VEL
LIN {X 0,Y 474.654,Z 414.363,A -85,B 0,C 180,E1 -7399.911,E2 -7399.911} C_VEL
LIN {X 0,Y 474.637,Z 414.361,A -85,B 0,C 180,E1 -7403.358,E2 -7403.358} C_VEL
LIN {X 0,Y 474.629,Z 414.359,A -85,B 0,C 180,E1 -7406.374,E2 -7406.374} C_VEL
LIN {X 0,Y 474.623,Z 414.366,A -85,B 0,C 180,E1 -7409.252,E2 -7409.252} C_VEL
LIN {X 0,Y 474.618,Z 414.357,A -85,B 0,C 180,E1 -7412.431,E2 -7412.431} C_VEL
LIN {X 0,Y 474.617,Z 414.364,A -85,B 0,C 180,E1 -7415.469,E2 -7415.469} C_VEL
LIN {X 0,Y 474.615,Z 414.364,A -85,B 0,C 180,E1 -7418.457,E2 -7418.457} C_VEL
LIN {X 0,Y 474.623,Z 414.36,A -85,B 0,C 180,E1 -7421.785,E2 -7421.785} C_VEL
LIN {X 0,Y 474.624,Z 414.365,A -85,B 0,C 180,E1 -7424.703,E2 -7424.703} C_VEL
LIN {X 0,Y 474.628,Z 414.36,A -85,B 0,C 180,E1 -7427.763,E2 -7427.763} C_VEL
LIN {X 0,Y 474.636,Z 414.359,A -85,B 0,C 180,E1 -7430.453,E2 -7430.453} C_VEL
LIN {X 0,Y 474.587,Z 414.364,A -85,B 0,C 180,E1 -7433.676,E2 -7433.676} C_VEL
LIN {X 0,Y 474.646,Z 414.363,A -85,B 0,C 180,E1 -7436.78,E2 -7436.78} C_VEL
LIN {X 0,Y 474.618,Z 414.363,A -85,B 0,C 180,E1 -7438,E2 -7438} C_VEL
LIN {X 0,Y 473.915,Z 414.456,A -85,B 0,C 180,E1 -7438.709,E2 -7438.709} C_VEL
LIN {X 0,Y 471.041,Z 414.812,A -85,B 0,C 180,E1 -7439.859,E2 -7439.859} C_VEL
LIN {X 0,Y 468.635,Z 415.114,A -85,B 0,C 180,E1 -7440.787,E2 -7440.787} C_VEL
LIN {X 0,Y 467.611,Z 415.239,A -85,B 0,C 180,E1 -7441.504,E2 -7441.504} C_VEL
LIN {X 0,Y 467.531,Z 415.25,A -85,B 0,C 180,E1 -7441.746,E2 -7441.746} C_VEL
LIN {X 0,Y 467.592,Z 415.318,A -85,B 0,C 180,E1 -7443.979,E2 -7443.979} C_VEL
LIN {X 0,Y 469.778,Z 426.019,A -85,B 0,C 180,E1 -7445.864,E2 -7445.864} C_VEL
LIN {X 0,Y 469.997,Z 430.69,A -85,B 0,C 180,E1 -7446.655,E2 -7446.655} C_VEL
LIN {X 0,Y 469.36,Z 448.789,A -85,B 0,C 180,E1 -7449.627,E2 -7449.627} C_VEL
LIN {X 0,Y 468.829,Z 467.361,A -85,B 0,C 180,E1 -7452.554,E2 -7452.554} C_VEL
LIN {X 0,Y 468.793,Z 470.626,A -85,B 0,C 180,E1 -7453.038,E2 -7453.038} C_VEL
LIN {X 0,Y 471.322,Z 485.465,A -85,B 0,C 180,E1 -7453.371,E2 -7453.371} C_VEL
LIN {X 0,Y 470.592,Z 578.974,A -85,B 0,C 180,E1 -7454.822,E2 -7454.822} C_VEL
LIN {X 0,Y 470.338,Z 591.97,A -85,B 0,C 180,E1 -7455.174,E2 -7455.174} C_VEL
LIN {X 0,Y 469.985,Z 603.948,A -85,B 0,C 180,E1 -7455.66,E2 -7455.66} C_VEL
LIN {X 0,Y 469.584,Z 614.948,A -85,B 0,C 180,E1 -7456.265,E2 -7456.265} C_VEL
LIN {X 0,Y 469.183,Z 625.619,A -85,B 0,C 180,E1 -7457.015,E2 -7457.015} C_VEL
LIN {X 0,Y 468.678,Z 636.693,A -85,B 0,C 180,E1 -7457.991,E2 -7457.991} C_VEL
LIN {X 0,Y 468.152,Z 645.669,A -85,B 0,C 180,E1 -7458.965,E2 -7458.965} C_VEL
LIN {X 0,Y 467.716,Z 655.313,A -85,B 0,C 180,E1 -7460.268,E2 -7460.268} C_VEL
LIN {X 0,Y 467.344,Z 663.069,A -85,B 0,C 180,E1 -7461.569,E2 -7461.569} C_VEL
LIN {X 0,Y 467.1,Z 668.311,A -85,B 0,C 180,E1 -7462.652,E2 -7462.652} C_VEL
LIN {X 0,Y 466.998,Z 673.433,A -85,B 0,C 180,E1 -7463.953,E2 -7463.953} C_VEL
LIN {X 0,Y 466.74,Z 677.406,A -85,B 0,C 180,E1 -7465.249,E2 -7465.249} C_VEL
LIN {X 0,Y 466.771,Z 680.332,A -85,B 0,C 180,E1 -7466.547,E2 -7466.547} C_VEL
LIN {X 0,Y 466.684,Z 681.757,A -85,B 0,C 180,E1 -7467.411,E2 -7467.411} C_VEL
LIN {X 0,Y 466.62,Z 683.37,A -85,B 0,C 180,E1 -7469.137,E2 -7469.137} C_VEL
LIN {X 0,Y 466.599,Z 683.607,A -85,B 0,C 180,E1 -7470,E2 -7470} C_VEL
LIN {X 0,Y 466.619,Z 683.419,A -85,B 0,C 180,E1 -7470.863,E2 -7470.863} C_VEL
LIN {X 0,Y 466.684,Z 681.871,A -85,B 0,C 180,E1 -7472.589,E2 -7472.589} C_VEL
LIN {X 0,Y 466.771,Z 680.509,A -85,B 0,C 180,E1 -7473.453,E2 -7473.453} C_VEL
LIN {X 0,Y 466.739,Z 677.649,A -85,B 0,C 180,E1 -7474.751,E2 -7474.751} C_VEL
LIN {X 0,Y 466.969,Z 673.756,A -85,B 0,C 180,E1 -7476.047,E2 -7476.047} C_VEL
LIN {X 0,Y 467.099,Z 668.717,A -85,B 0,C 180,E1 -7477.348,E2 -7477.348} C_VEL
LIN {X 0,Y 467.376,Z 662.362,A -85,B 0,C 180,E1 -7478.648,E2 -7478.648} C_VEL
LIN {X 0,Y 467.74,Z 654.468,A -85,B 0,C 180,E1 -7479.95,E2 -7479.95} C_VEL
LIN {X 0,Y 468.13,Z 646.405,A -85,B 0,C 180,E1 -7481.035,E2 -7481.035} C_VEL
LIN {X 0,Y 468.706,Z 636.504,A -85,B 0,C 180,E1 -7482.118,E2 -7482.118} C_VEL
LIN {X 0,Y 469.179,Z 625.289,A -85,B 0,C 180,E1 -7483.102,E2 -7483.102} C_VEL
LIN {X 0,Y 469.622,Z 614.51,A -85,B 0,C 180,E1 -7483.854,E2 -7483.854} C_VEL
LIN {X 0,Y 470.011,Z 603.543,A -85,B 0,C 180,E1 -7484.449,E2 -7484.449} C_VEL
LIN {X 0,Y 470.377,Z 590.557,A -85,B 0,C 180,E1 -7484.964,E2 -7484.964} C_VEL
LIN {X 0,Y 470.667,Z 578.061,A -85,B 0,C 180,E1 -7485.286,E2 -7485.286} C_VEL
LIN {X 0,Y 471.225,Z 484.966,A -85,B 0,C 180,E1 -7486.731,E2 -7486.731} C_VEL
LIN {X 0,Y 468.797,Z 470.58,A -85,B 0,C 180,E1 -7487.059,E2 -7487.059} C_VEL
LIN {X 0,Y 469.223,Z 453.635,A -85,B 0,C 180,E1 -7489.694,E2 -7489.694} C_VEL
LIN {X 0,Y 469.855,Z 435.5,A -85,B 0,C 180,E1 -7492.654,E2 -7492.654} C_VEL
LIN {X 0,Y 469.963,Z 427.367,A -85,B 0,C 180,E1 -7494.003,E2 -7494.003} C_VEL
LIN {X 0,Y 467.558,Z 415.248,A -85,B 0,C 180,E1 -7496.143,E2 -7496.143} C_VEL
LIN {X 0,Y 467.553,Z 415.247,A -85,B 0,C 180,E1 -7499.328,E2 -7499.328} C_VEL
LIN {X 0,Y 467.585,Z 415.241,A -85,B 0,C 180,E1 -7502.679,E2 -7502.679} C_VEL
LIN {X 0,Y 467.56,Z 415.246,A -85,B 0,C 180,E1 -7505.739,E2 -7505.739} C_VEL
LIN {X 0,Y 467.578,Z 415.245,A -85,B 0,C 180,E1 -7509.145,E2 -7509.145} C_VEL
LIN {X 0,Y 467.589,Z 415.239,A -85,B 0,C 180,E1 -7512.567,E2 -7512.567} C_VEL
LIN {X 0,Y 467.574,Z 415.244,A -85,B 0,C 180,E1 -7515.053,E2 -7515.053} C_VEL
LIN {X 0,Y 467.592,Z 415.235,A -85,B 0,C 180,E1 -7517.44,E2 -7517.44} C_VEL
LIN {X 0,Y 467.585,Z 415.245,A -85,B 0,C 180,E1 -7520.855,E2 -7520.855} C_VEL
LIN {X 0,Y 467.56,Z 415.235,A -85,B 0,C 180,E1 -7524.261,E2 -7524.261} C_VEL
LIN {X 0,Y 467.585,Z 415.238,A -85,B 0,C 180,E1 -7527.321,E2 -7527.321} C_VEL
LIN {X 0,Y 467.553,Z 415.247,A -85,B 0,C 180,E1 -7530.672,E2 -7530.672} C_VEL
LIN {X 0,Y 467.564,Z 415.243,A -85,B 0,C 180,E1 -7533.678,E2 -7533.678} C_VEL
LIN {X 0,Y 467.598,Z 415.383,A -85,B 0,C 180,E1 -7534.01,E2 -7534.01} C_VEL
LIN {X 0,Y 470.01,Z 428.011,A -85,B 0,C 180,E1 -7536.188,E2 -7536.188} C_VEL
LIN {X 0,Y 469.68,Z 442.405,A -85,B 0,C 180,E1 -7538.506,E2 -7538.506} C_VEL
LIN {X 0,Y 469.106,Z 460.613,A -85,B 0,C 180,E1 -7541.436,E2 -7541.436} C_VEL
LIN {X 0,Y 468.821,Z 471.277,A -85,B 0,C 180,E1 -7543.116,E2 -7543.116} C_VEL
LIN {X 0,Y 471.126,Z 486.194,A -85,B 0,C 180,E1 -7543.457,E2 -7543.457} C_VEL
LIN {X 0,Y 470.152,Z 581.455,A -85,B 0,C 180,E1 -7545.085,E2 -7545.085} C_VEL
LIN {X 0,Y 469.789,Z 595.328,A -85,B 0,C 180,E1 -7545.516,E2 -7545.516} C_VEL
LIN {X 0,Y 469.479,Z 606.788,A -85,B 0,C 180,E1 -7546.031,E2 -7546.031} C_VEL
LIN {X 0,Y 469.014,Z 619.399,A -85,B 0,C 180,E1 -7546.791,E2 -7546.791} C_VEL
LIN {X 0,Y 468.682,Z 630.859,A -85,B 0,C 180,E1 -7547.68,E2 -7547.68} C_VEL
LIN {X 0,Y 468.12,Z 641.766,A -85,B 0,C 180,E1 -7548.745,E2 -7548.745} C_VEL
LIN {X 0,Y 467.793,Z 650.785,A -85,B 0,C 180,E1 -7549.832,E2 -7549.832} C_VEL
LIN {X 0,Y 467.383,Z 659.484,A -85,B 0,C 180,E1 -7551.134,E2 -7551.134} C_VEL
LIN {X 0,Y 467.067,Z 666.502,A -85,B 0,C 180,E1 -7552.434,E2 -7552.434} C_VEL
LIN {X 0,Y 466.922,Z 671.902,A -85,B 0,C 180,E1 -7553.687,E2 -7553.687} C_VEL
LIN {X 0,Y 466.797,Z 675.785,A -85,B 0,C 180,E1 -7554.817,E2 -7554.817} C_VEL
LIN {X 0,Y 466.737,Z 678.176,A -85,B 0,C 180,E1 -7555.682,E2 -7555.682} C_VEL
LIN {X 0,Y 466.767,Z 680.112,A -85,B 0,C 180,E1 -7556.547,E2 -7556.547} C_VEL
LIN {X 0,Y 466.683,Z 681.636,A -85,B 0,C 180,E1 -7557.411,E2 -7557.411} C_VEL
LIN {X 0,Y 466.635,Z 682.692,A -85,B 0,C 180,E1 -7558.274,E2 -7558.274} C_VEL
LIN {X 0,Y 466.62,Z 683.347,A -85,B 0,C 180,E1 -7559.137,E2 -7559.137} C_VEL
LIN {X 0,Y 466.599,Z 683.611,A -85,B 0,C 180,E1 -7560,E2 -7560} C_VEL
LIN {X 0,Y 466.619,Z 683.427,A -85,B 0,C 180,E1 -7560.863,E2 -7560.863} C_VEL
LIN {X 0,Y 466.683,Z 681.85,A -85,B 0,C 180,E1 -7562.589,E2 -7562.589} C_VEL
LIN {X 0,Y 466.767,Z 680.412,A -85,B 0,C 180,E1 -7563.453,E2 -7563.453} C_VEL
LIN {X 0,Y 466.729,Z 677.437,A -85,B 0,C 180,E1 -7564.751,E2 -7564.751} C_VEL
LIN {X 0,Y 466.942,Z 673.378,A -85,B 0,C 180,E1 -7566.048,E2 -7566.048} C_VEL
LIN {X 0,Y 467.096,Z 667.152,A -85,B 0,C 180,E1 -7567.565,E2 -7567.565} C_VEL
LIN {X 0,Y 467.368,Z 660.259,A -85,B 0,C 180,E1 -7568.867,E2 -7568.867} C_VEL
LIN {X 0,Y 467.742,Z 651.677,A -85,B 0,C 180,E1 -7570.169,E2 -7570.169} C_VEL
LIN {X 0,Y 468.099,Z 642.841,A -85,B 0,C 180,E1 -7571.255,E2 -7571.255} C_VEL
LIN {X 0,Y 468.617,Z 632.222,A -85,B 0,C 180,E1 -7572.309,E2 -7572.309} C_VEL
LIN {X 0,Y 468.997,Z 621.232,A -85,B 0,C 180,E1 -7573.188,E2 -7573.188} C_VEL
LIN {X 0,Y 469.381,Z 608.58,A -85,B 0,C 180,E1 -7573.971,E2 -7573.971} C_VEL
LIN {X 0,Y 469.805,Z 597.039,A -85,B 0,C 180,E1 -7574.511,E2 -7574.511} C_VEL
LIN {X 0,Y 470.073,Z 583.805,A -85,B 0,C 180,E1 -7574.946,E2 -7574.946} C_VEL
LIN {X 0,Y 470.353,Z 567.08,A -85,B 0,C 180,E1 -7575.269,E2 -7575.269} C_VEL
LIN {X 0,Y 471.265,Z 485.154,A -85,B 0,C 180,E1 -7576.719,E2 -7576.719} C_VEL
LIN {X 0,Y 469.001,Z 471.806,A -85,B 0,C 180,E1 -7577.086,E2 -7577.086} C_VEL
LIN {X 0,Y 469.508,Z 452.311,A -85,B 0,C 180,E1 -7580.138,E2 -7580.138} C_VEL
LIN {X 0,Y 470.008,Z 434.595,A -85,B 0,C 180,E1 -7582.878,E2 -7582.878} C_VEL
LIN {X 0,Y 470.074,Z 427.529,A -85,B 0,C 180,E1 -7583.984,E2 -7583.984} C_VEL
LIN {X 0,Y 467.579,Z 415.245,A -85,B 0,C 180,E1 -7586.051,E2 -7586.051} C_VEL
LIN {X 0,Y 467.553,Z 415.249,A -85,B 0,C 180,E1 -7589.328,E2 -7589.328} C_VEL
LIN {X 0,Y 467.584,Z 415.24,A -85,B 0,C 180,E1 -7592.679,E2 -7592.679} C_VEL
LIN {X 0,Y 467.56,Z 415.245,A -85,B 0,C 180,E1 -7595.739,E2 -7595.739} C_VEL
LIN {X 0,Y 467.584,Z 415.243,A -85,B 0,C 180,E1 -7599.145,E2 -7599.145} C_VEL
LIN {X 0,Y 467.589,Z 415.24,A -85,B 0,C 180,E1 -7602.567,E2 -7602.567} C_VEL
LIN {X 0,Y 467.573,Z 415.243,A -85,B 0,C 180,E1 -7605.053,E2 -7605.053} C_VEL
LIN {X 0,Y 467.591,Z 415.24,A -85,B 0,C 180,E1 -7607.44,E2 -7607.44} C_VEL
LIN {X 0,Y 467.584,Z 415.24,A -85,B 0,C 180,E1 -7610.855,E2 -7610.855} C_VEL
LIN {X 0,Y 467.56,Z 415.244,A -85,B 0,C 180,E1 -7614.261,E2 -7614.261} C_VEL
LIN {X 0,Y 467.584,Z 415.239,A -85,B 0,C 180,E1 -7617.321,E2 -7617.321} C_VEL
LIN {X 0,Y 467.552,Z 415.248,A -85,B 0,C 180,E1 -7620.672,E2 -7620.672} C_VEL
LIN {X 0,Y 467.625,Z 415.409,A -85,B 0,C 180,E1 -7621.254,E2 -7621.254} C_VEL
LIN {X 0,Y 470.812,Z 430.763,A -85,B 0,C 180,E1 -7623.784,E2 -7623.784} C_VEL
LIN {X 0,Y 470.281,Z 445.128,A -85,B 0,C 180,E1 -7625.948,E2 -7625.948} C_VEL
LIN {X 0,Y 469.386,Z 465.319,A -85,B 0,C 180,E1 -7628.94,E2 -7628.94} C_VEL
LIN {X 0,Y 468.56,Z 488.32,A -85,B 0,C 180,E1 -7632.318,E2 -7632.318} C_VEL
LIN {X 0,Y 468.371,Z 493.105,A -85,B 0,C 180,E1 -7633.006,E2 -7633.006} C_VEL
LIN {X 0,Y 470.993,Z 514.444,A -85,B 0,C 180,E1 -7633.469,E2 -7633.469} C_VEL
LIN {X 0,Y 469.988,Z 606.956,A -85,B 0,C 180,E1 -7635.052,E2 -7635.052} C_VEL
LIN {X 0,Y 469.719,Z 619.079,A -85,B 0,C 180,E1 -7635.403,E2 -7635.403} C_VEL
LIN {X 0,Y 469.241,Z 632.304,A -85,B 0,C 180,E1 -7635.969,E2 -7635.969} C_VEL
LIN {X 0,Y 468.885,Z 644.172,A -85,B 0,C 180,E1 -7636.676,E2 -7636.676} C_VEL
LIN {X 0,Y 468.406,Z 655.836,A -85,B 0,C 180,E1 -7637.571,E2 -7637.571} C_VEL
LIN {X 0,Y 467.99,Z 665.738,A -85,B 0,C 180,E1 -7638.523,E2 -7638.523} C_VEL
LIN {X 0,Y 467.545,Z 674.882,A -85,B 0,C 180,E1 -7639.608,E2 -7639.608} C_VEL
LIN {X 0,Y 467.199,Z 683.764,A -85,B 0,C 180,E1 -7640.912,E2 -7640.912} C_VEL
LIN {X 0,Y 466.982,Z 690.882,A -85,B 0,C 180,E1 -7642.215,E2 -7642.215} C_VEL
LIN {X 0,Y 466.814,Z 696.619,A -85,B 0,C 180,E1 -7643.54,E2 -7643.54} C_VEL
LIN {X 0,Y 466.776,Z 700.96,A -85,B 0,C 180,E1 -7644.817,E2 -7644.817} C_VEL
LIN {X 0,Y 466.728,Z 703.288,A -85,B 0,C 180,E1 -7645.682,E2 -7645.682} C_VEL
LIN {X 0,Y 466.805,Z 705.188,A -85,B 0,C 180,E1 -7646.547,E2 -7646.547} C_VEL
LIN {X 0,Y 466.718,Z 706.619,A -85,B 0,C 180,E1 -7647.411,E2 -7647.411} C_VEL
LIN {X 0,Y 466.667,Z 708.245,A -85,B 0,C 180,E1 -7649.137,E2 -7649.137} C_VEL
LIN {X 0,Y 466.656,Z 708.468,A -85,B 0,C 180,E1 -7650,E2 -7650} C_VEL
LIN {X 0,Y 466.666,Z 708.258,A -85,B 0,C 180,E1 -7650.863,E2 -7650.863} C_VEL
LIN {X 0,Y 466.72,Z 706.62,A -85,B 0,C 180,E1 -7652.589,E2 -7652.589} C_VEL
LIN {X 0,Y 466.817,Z 705.19,A -85,B 0,C 180,E1 -7653.452,E2 -7653.452} C_VEL
LIN {X 0,Y 466.734,Z 702.203,A -85,B 0,C 180,E1 -7654.751,E2 -7654.751} C_VEL
LIN {X 0,Y 466.783,Z 698.15,A -85,B 0,C 180,E1 -7656.05,E2 -7656.05} C_VEL
LIN {X 0,Y 466.968,Z 691.897,A -85,B 0,C 180,E1 -7657.567,E2 -7657.567} C_VEL
LIN {X 0,Y 467.195,Z 685.07,A -85,B 0,C 180,E1 -7658.87,E2 -7658.87} C_VEL
LIN {X 0,Y 467.436,Z 678.077,A -85,B 0,C 180,E1 -7659.957,E2 -7659.957} C_VEL
LIN {X 0,Y 467.788,Z 669.623,A -85,B 0,C 180,E1 -7661.044,E2 -7661.044} C_VEL
LIN {X 0,Y 468.23,Z 659.146,A -85,B 0,C 180,E1 -7662.13,E2 -7662.13} C_VEL
LIN {X 0,Y 468.652,Z 648.751,A -85,B 0,C 180,E1 -7663,E2 -7663} C_VEL
LIN {X 0,Y 469.115,Z 637.262,A -85,B 0,C 180,E1 -7663.759,E2 -7663.759} C_VEL
LIN {X 0,Y 469.522,Z 625.291,A -85,B 0,C 180,E1 -7664.354,E2 -7664.354} C_VEL
LIN {X 0,Y 469.88,Z 612.286,A -85,B 0,C 180,E1 -7664.813,E2 -7664.813} C_VEL
LIN {X 0,Y 470.107,Z 599.769,A -85,B 0,C 180,E1 -7665.083,E2 -7665.083} C_VEL
LIN {X 0,Y 470.556,Z 551.306,A -85,B 0,C 180,E1 -7665.87,E2 -7665.87} C_VEL
LIN {X 0,Y 470.83,Z 512.489,A -85,B 0,C 180,E1 -7666.569,E2 -7666.569} C_VEL
LIN {X 0,Y 468.214,Z 489.641,A -85,B 0,C 180,E1 -7667.115,E2 -7667.115} C_VEL
LIN {X 0,Y 468.917,Z 467.244,A -85,B 0,C 180,E1 -7670.394,E2 -7670.394} C_VEL
LIN {X 0,Y 469.622,Z 448.933,A -85,B 0,C 180,E1 -7673.131,E2 -7673.131} C_VEL
LIN {X 0,Y 470.531,Z 430.364,A -85,B 0,C 180,E1 -7675.978,E2 -7675.978} C_VEL
LIN {X 0,Y 469.096,Z 421.838,A -85,B 0,C 180,E1 -7677.432,E2 -7677.432} C_VEL
LIN {X 0,Y 467.608,Z 415.24,A -85,B 0,C 180,E1 -7678.625,E2 -7678.625} C_VEL
LIN {X 0,Y 467.584,Z 415.245,A -85,B 0,C 180,E1 -7681.74,E2 -7681.74} C_VEL
LIN {X 0,Y 467.564,Z 415.243,A -85,B 0,C 180,E1 -7684.833,E2 -7684.833} C_VEL
LIN {X 0,Y 467.564,Z 415.243,A -85,B 0,C 180,E1 -7688.045,E2 -7688.045} C_VEL
LIN {X 0,Y 467.577,Z 415.244,A -85,B 0,C 180,E1 -7691.276,E2 -7691.276} C_VEL
LIN {X 0,Y 467.551,Z 415.245,A -85,B 0,C 180,E1 -7693.82,E2 -7693.82} C_VEL
LIN {X 0,Y 467.558,Z 415.242,A -85,B 0,C 180,E1 -7696.256,E2 -7696.256} C_VEL
LIN {X 0,Y 467.58,Z 415.24,A -85,B 0,C 180,E1 -7698.723,E2 -7698.723} C_VEL
LIN {X 0,Y 467.567,Z 415.241,A -85,B 0,C 180,E1 -7701.956,E2 -7701.956} C_VEL
LIN {X 0,Y 467.568,Z 415.244,A -85,B 0,C 180,E1 -7705.168,E2 -7705.168} C_VEL
LIN {X 0,Y 467.586,Z 415.24,A -85,B 0,C 180,E1 -7708.26,E2 -7708.26} C_VEL
LIN {X 0,Y 467.578,Z 415.243,A -85,B 0,C 180,E1 -7711.25,E2 -7711.25} C_VEL
LIN {X 0,Y 467.6,Z 415.24,A -85,B 0,C 180,E1 -7714.159,E2 -7714.159} C_VEL
LIN {X 0,Y 467.579,Z 415.245,A -85,B 0,C 180,E1 -7716.996,E2 -7716.996} C_VEL
LIN {X 0,Y 467.625,Z 415.236,A -85,B 0,C 180,E1 -7719.777,E2 -7719.777} C_VEL
LIN {X 0,Y 467.607,Z 415.24,A -85,B 0,C 180,E1 -7723.024,E2 -7723.024} C_VEL
LIN {X 0,Y 471.612,Z 426.565,A -85,B 0,C 180,E1 -7723.427,E2 -7723.427} C_VEL
LIN {X 0,Y 470.349,Z 518.024,A -85,B 0,C 180,E1 -7725.091,E2 -7725.091} C_VEL
LIN {X 0,Y 470.167,Z 531.163,A -85,B 0,C 180,E1 -7725.5,E2 -7725.5} C_VEL
LIN {X 0,Y 469.918,Z 543.257,A -85,B 0,C 180,E1 -7726.045,E2 -7726.045} C_VEL
LIN {X 0,Y 469.551,Z 555.191,A -85,B 0,C 180,E1 -7726.768,E2 -7726.768} C_VEL
LIN {X 0,Y 469.122,Z 566.839,A -85,B 0,C 180,E1 -7727.674,E2 -7727.674} C_VEL
LIN {X 0,Y 468.77,Z 575.817,A -85,B 0,C 180,E1 -7728.542,E2 -7728.542} C_VEL
LIN {X 0,Y 468.359,Z 584.995,A -85,B 0,C 180,E1 -7729.626,E2 -7729.626} C_VEL
LIN {X 0,Y 467.955,Z 593.864,A -85,B 0,C 180,E1 -7730.927,E2 -7730.927} C_VEL
LIN {X 0,Y 467.625,Z 600.969,A -85,B 0,C 180,E1 -7732.226,E2 -7732.226} C_VEL
LIN {X 0,Y 467.432,Z 606.58,A -85,B 0,C 180,E1 -7733.525,E2 -7733.525} C_VEL
LIN {X 0,Y 467.174,Z 610.974,A -85,B 0,C 180,E1 -7734.821,E2 -7734.821} C_VEL
LIN {X 0,Y 467.2,Z 613.258,A -85,B 0,C 180,E1 -7735.687,E2 -7735.687} C_VEL
LIN {X 0,Y 467.032,Z 615.136,A -85,B 0,C 180,E1 -7736.549,E2 -7736.549} C_VEL
LIN {X 0,Y 466.872,Z 616.569,A -85,B 0,C 180,E1 -7737.412,E2 -7737.412} C_VEL
LIN {X 0,Y 466.755,Z 618.13,A -85,B 0,C 180,E1 -7739.137,E2 -7739.137} C_VEL
LIN {X 0,Y 466.745,Z 618.318,A -85,B 0,C 180,E1 -7740,E2 -7740} C_VEL
LIN {X 0,Y 466.746,Z 618.069,A -85,B 0,C 180,E1 -7740.863,E2 -7740.863} C_VEL
LIN {X 0,Y 466.857,Z 616.348,A -85,B 0,C 180,E1 -7742.588,E2 -7742.588} C_VEL
LIN {X 0,Y 467.028,Z 614.875,A -85,B 0,C 180,E1 -7743.451,E2 -7743.451} C_VEL
LIN {X 0,Y 467.11,Z 611.836,A -85,B 0,C 180,E1 -7744.747,E2 -7744.747} C_VEL
LIN {X 0,Y 467.243,Z 606.566,A -85,B 0,C 180,E1 -7746.354,E2 -7746.354} C_VEL
LIN {X 0,Y 467.466,Z 600.392,A -85,B 0,C 180,E1 -7747.777,E2 -7747.777} C_VEL
LIN {X 0,Y 467.806,Z 593.237,A -85,B 0,C 180,E1 -7749.076,E2 -7749.076} C_VEL
LIN {X 0,Y 468.166,Z 584.286,A -85,B 0,C 180,E1 -7750.378,E2 -7750.378} C_VEL
LIN {X 0,Y 468.594,Z 575.095,A -85,B 0,C 180,E1 -7751.462,E2 -7751.462} C_VEL
LIN {X 0,Y 468.998,Z 564.891,A -85,B 0,C 180,E1 -7752.44,E2 -7752.44} C_VEL
LIN {X 0,Y 469.376,Z 553.962,A -85,B 0,C 180,E1 -7753.281,E2 -7753.281} C_VEL
LIN {X 0,Y 469.704,Z 541.835,A -85,B 0,C 180,E1 -7754.017,E2 -7754.017} C_VEL
LIN {X 0,Y 470.016,Z 529.087,A -85,B 0,C 180,E1 -7754.588,E2 -7754.588} C_VEL
LIN {X 0,Y 470.25,Z 515.723,A -85,B 0,C 180,E1 -7754.995,E2 -7754.995} C_VEL
LIN {X 0,Y 471.221,Z 425.929,A -85,B 0,C 180,E1 -7756.536,E2 -7756.536} C_VEL
LIN {X 0,Y 467.606,Z 415.239,A -85,B 0,C 180,E1 -7756.857,E2 -7756.857} C_VEL
LIN {X 0,Y 467.623,Z 415.242,A -85,B 0,C 180,E1 -7759.308,E2 -7759.308} C_VEL
LIN {X 0,Y 467.537,Z 415.243,A -85,B 0,C 180,E1 -7762.074,E2 -7762.074} C_VEL
LIN {X 0,Y 467.571,Z 415.24,A -85,B 0,C 180,E1 -7764.889,E2 -7764.889} C_VEL
LIN {X 0,Y 467.618,Z 415.232,A -85,B 0,C 180,E1 -7767.769,E2 -7767.769} C_VEL
LIN {X 0,Y 467.571,Z 415.245,A -85,B 0,C 180,E1 -7771.045,E2 -7771.045} C_VEL
LIN {X 0,Y 467.591,Z 415.226,A -85,B 0,C 180,E1 -7774.242,E2 -7774.242} C_VEL
LIN {X 0,Y 467.551,Z 415.248,A -85,B 0,C 180,E1 -7777.186,E2 -7777.186} C_VEL
LIN {X 0,Y 467.577,Z 415.233,A -85,B 0,C 180,E1 -7780.265,E2 -7780.265} C_VEL
LIN {X 0,Y 467.589,Z 415.24,A -85,B 0,C 180,E1 -7782.567,E2 -7782.567} C_VEL
LIN {X 0,Y 467.573,Z 415.236,A -85,B 0,C 180,E1 -7785.053,E2 -7785.053} C_VEL
LIN {X 0,Y 467.592,Z 415.238,A -85,B 0,C 180,E1 -7787.44,E2 -7787.44} C_VEL
LIN {X 0,Y 467.578,Z 415.243,A -85,B 0,C 180,E1 -7790.855,E2 -7790.855} C_VEL
LIN {X 0,Y 467.56,Z 415.243,A -85,B 0,C 180,E1 -7794.261,E2 -7794.261} C_VEL
LIN {X 0,Y 467.585,Z 415.239,A -85,B 0,C 180,E1 -7797.321,E2 -7797.321} C_VEL
LIN {X 0,Y 467.553,Z 415.25,A -85,B 0,C 180,E1 -7800.672,E2 -7800.672} C_VEL
LIN {X 0,Y 467.531,Z 415.25,A -85,B 0,C 180,E1 -7801.746,E2 -7801.746} C_VEL
LIN {X 0,Y 466.84,Z 415.347,A -85,B 0,C 180,E1 -7802.245,E2 -7802.245} C_VEL
LIN {X 0,Y 463.982,Z 415.694,A -85,B 0,C 180,E1 -7803.03,E2 -7803.03} C_VEL
LIN {X 0,Y 461.783,Z 416.612,A -85,B 0,C 180,E1 -7803.631,E2 -7803.631} C_VEL
LIN {X 0,Y 461.02,Z 418.063,A -85,B 0,C 180,E1 -7804.073,E2 -7804.073} C_VEL
